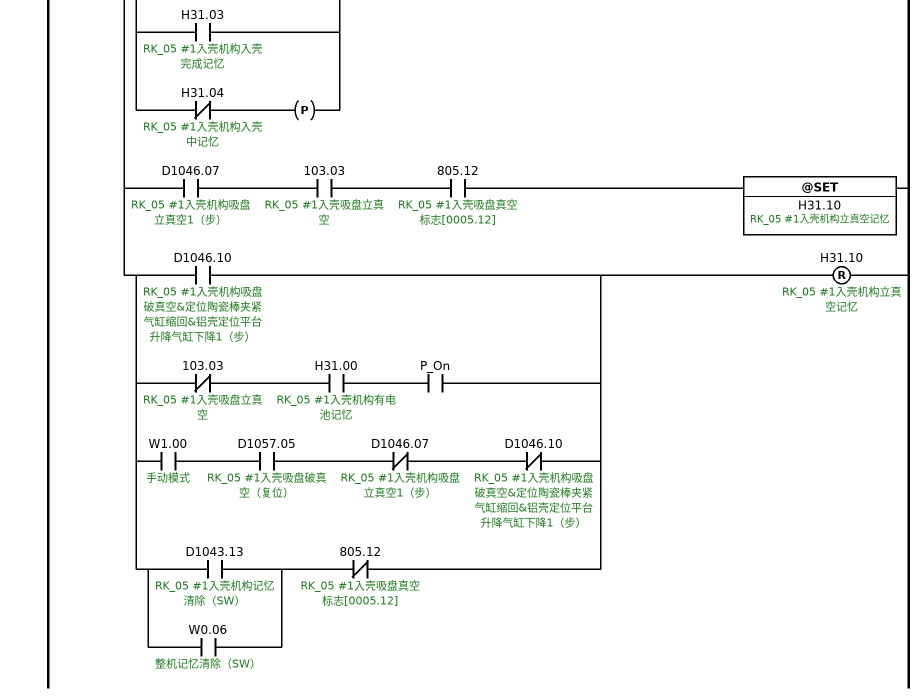
; [picture p456: 入壳_RK_05 / 自动_1入壳, rungs 30-30]
; rung 30: #1入壳机构记忆
LD P_On
OUT TR0
AND H31.03  ; RK_05 #1入壳机构入壳完成记忆
@SET H31.00  ; RK_05 #1入壳机构有电池记忆
LD TR0
LD D1092.03  ; RK_06 电池上下料机构电池下料夹爪气缸夹紧3（步）
AND H40.00  ; RK_06 U8_X 电池上下料X轴回原点记忆
AND 863.04  ; RK_06 U8_X 电池上下料X轴#1入壳取料位标志
AND 814.02  ; RK_06 电池下料升降气缸下降位标志[0014.02]
LD D1043.13  ; RK_05 #1入壳机构记忆清除（SW）
OR W0.06  ; 整机记忆清除（SW）
LDNOT 805.09  ; RK_05 #1入壳铝壳有料感应标志[0005.09]
LD H7.15  ; 空跑程序
AND 5.09  ; RK_05 #1入壳铝壳有料感应
ORLD
ANDLD
ORLD
ANDLD
RSET H31.00  ; RK_05 #1入壳机构有电池记忆
LD TR0
AND D1026.10  ; RK_03 电芯上料机构上料夹爪气缸张开（步）
LD H20.00  ; RK_03 U0_U 电芯上料X轴回原点记忆
AND 853.02  ; RK_03 U0_U 电芯上料X轴#1入壳放料位标志
AND 800.08  ; RK_03 电芯上料升降气缸下降位标志[0000.08]
LD 805.08  ; RK_05 #1入壳电芯有料感应标志[0005.08]
ANDNOT P_On
ORLD
ANDLD
@SET H31.01  ; RK_05 #1入壳机构有电芯记忆
LD TR0
LD H31.03  ; RK_05 #1入壳机构入壳完成记忆
LDNOT H31.04  ; RK_05 #1入壳机构入壳中记忆
ANDNOT 805.08  ; RK_05 #1入壳电芯有料感应标志[0005.08]
ANDNOT P_On
ORLD
LD D1043.13  ; RK_05 #1入壳机构记忆清除（SW）
OR W0.06  ; 整机记忆清除（SW）
LDNOT H31.04  ; RK_05 #1入壳机构入壳中记忆
ANDNOT 805.08  ; RK_05 #1入壳电芯有料感应标志[0005.08]
AND P_On
LD H7.15  ; 空跑程序
ANDNOT 5.08  ; RK_05 #1入壳电芯有料感应
ORLD
ANDLD
ORLD
ANDLD
RSET H31.01  ; RK_05 #1入壳机构有电芯记忆
LD TR0
AND D1089.03  ; RK_06 电池上下料机构铝壳上料夹爪气缸张开2（步）
LD H40.00  ; RK_06 U8_X 电池上下料X轴回原点记忆
AND 863.02  ; RK_06 U8_X 电池上下料X轴#1入壳放料位标志
AND 814.00  ; RK_06 铝壳上料升降气缸下降位标志[0014.00]
LD 805.09  ; RK_05 #1入壳铝壳有料感应标志[0005.09]
ANDNOT H31.00  ; RK_05 #1入壳机构有电池记忆
ORLD
ANDLD
@SET H31.02  ; RK_05 #1入壳机构有铝壳记忆
LD TR0
LD H31.03  ; RK_05 #1入壳机构入壳完成记忆
LD D1043.13  ; RK_05 #1入壳机构记忆清除（SW）
OR W0.06  ; 整机记忆清除（SW）
LDNOT 805.09  ; RK_05 #1入壳铝壳有料感应标志[0005.09]
LD H7.15  ; 空跑程序
AND 5.09  ; RK_05 #1入壳铝壳有料感应
ORLD
ANDLD
ORLD
ANDLD
RSET H31.02  ; RK_05 #1入壳机构有铝壳记忆
LD TR0
AND D1049.08  ; RK_05 #1入壳机构Y轴入壳位2（步）
AND 854.03  ; RK_05 U2_X #1入壳Y轴入壳位标志
AND H30.00  ; RK_05 U2_X #1入壳Y轴回原点记忆
ANDNOT W421.00  ; RK_05 #1入壳压力高[alm]
@SET H31.03  ; RK_05 #1入壳机构入壳完成记忆
LD TR0
LD H31.00  ; RK_05 #1入壳机构有电池记忆
LD D1043.13  ; RK_05 #1入壳机构记忆清除（SW）
OR W0.06  ; 整机记忆清除（SW）
LDNOT 805.09  ; RK_05 #1入壳铝壳有料感应标志[0005.09]
LD H7.15  ; 空跑程序
AND 5.09  ; RK_05 #1入壳铝壳有料感应
ORLD
ANDLD
ORLD
ANDLD
RSET H31.03  ; RK_05 #1入壳机构入壳完成记忆
LD TR0
AND D1049.02  ; RK_05 #1入壳机构Y轴电芯定位夹爪气缸松开位2（步）
@SET H31.04  ; RK_05 #1入壳机构入壳中记忆
LD TR0
LD H31.03  ; RK_05 #1入壳机构入壳完成记忆
LD D1043.13  ; RK_05 #1入壳机构记忆清除（SW）
OR W0.06  ; 整机记忆清除（SW）
LDNOT 805.09  ; RK_05 #1入壳铝壳有料感应标志[0005.09]
LD H7.15  ; 空跑程序
AND 5.09  ; RK_05 #1入壳铝壳有料感应
ORLD
ANDLD
ORLD
ANDLD
RSET H31.04  ; RK_05 #1入壳机构入壳中记忆
LD TR0
AND D1049.04  ; RK_05 #1入壳机构Y轴滚轮压紧位2（步）
AND 854.01  ; RK_05 U2_X #1入壳Y轴滚轮压紧位标志
@SET H31.06  ; RK_05 #1入壳机构Y轴滚轮压紧位记忆
LD TR0
LD D1049.06  ; RK_05 #1入壳机构Y轴滚轮松开位2（步）
OR H31.03  ; RK_05 #1入壳机构入壳完成记忆
ORNOT H31.04  ; RK_05 #1入壳机构入壳中记忆
ANDLD
RSET H31.06  ; RK_05 #1入壳机构Y轴滚轮压紧位记忆
LD TR0
AND D1049.06  ; RK_05 #1入壳机构Y轴滚轮松开位2（步）
AND 854.02  ; RK_05 U2_X #1入壳Y轴滚轮松开位标志
@SET H31.07  ; RK_05 #1入壳机构Y轴滚轮松开位记忆
LD TR0
LD H31.03  ; RK_05 #1入壳机构入壳完成记忆
ORNOT H31.04  ; RK_05 #1入壳机构入壳中记忆
ANDLD
RSET H31.07  ; RK_05 #1入壳机构Y轴滚轮松开位记忆
LD TR0
AND D1049.02  ; RK_05 #1入壳机构Y轴电芯定位夹爪气缸松开位2（步）
AND 854.04  ; RK_05 U2_X #1入壳Y轴电芯定位夹爪松开位标志
@SET H31.09  ; RK_05 #1入壳机构Y轴电芯定位夹爪松开位记忆
LD TR0
LD D1049.04  ; RK_05 #1入壳机构Y轴滚轮压紧位2（步）
OR H31.06  ; RK_05 #1入壳机构Y轴滚轮压紧位记忆
OR H31.03  ; RK_05 #1入壳机构入壳完成记忆
LDNOT H31.04  ; RK_05 #1入壳机构入壳中记忆
UP(521)
ORLD
ANDLD
RSET H31.09  ; RK_05 #1入壳机构Y轴电芯定位夹爪松开位记忆
LD TR0
AND D1046.07  ; RK_05 #1入壳机构吸盘立真空1（步）
AND 103.03  ; RK_05 #1入壳吸盘立真空
AND 805.12  ; RK_05 #1入壳吸盘真空标志[0005.12]
@SET H31.10  ; RK_05 #1入壳机构立真空记忆
LD TR0
LD D1046.10  ; RK_05 #1入壳机构吸盘破真空&定位陶瓷棒夹紧气缸缩回&铝壳定位平台升降气缸下降1（步）
LDNOT 103.03  ; RK_05 #1入壳吸盘立真空
AND H31.00  ; RK_05 #1入壳机构有电池记忆
AND P_On
ORLD
LD W1.00  ; 手动模式  // 20181116新增
AND D1057.05  ; RK_05 #1入壳吸盘破真空（复位）
ANDNOT D1046.07  ; RK_05 #1入壳机构吸盘立真空1（步）
ANDNOT D1046.10  ; RK_05 #1入壳机构吸盘破真空&定位陶瓷棒夹紧气缸缩回&铝壳定位平台升降气缸下降1（步）
ORLD
LD D1043.13  ; RK_05 #1入壳机构记忆清除（SW）
OR W0.06  ; 整机记忆清除（SW）
ANDNOT 805.12  ; RK_05 #1入壳吸盘真空标志[0005.12]
ORLD
ANDLD
RSET H31.10  ; RK_05 #1入壳机构立真空记忆

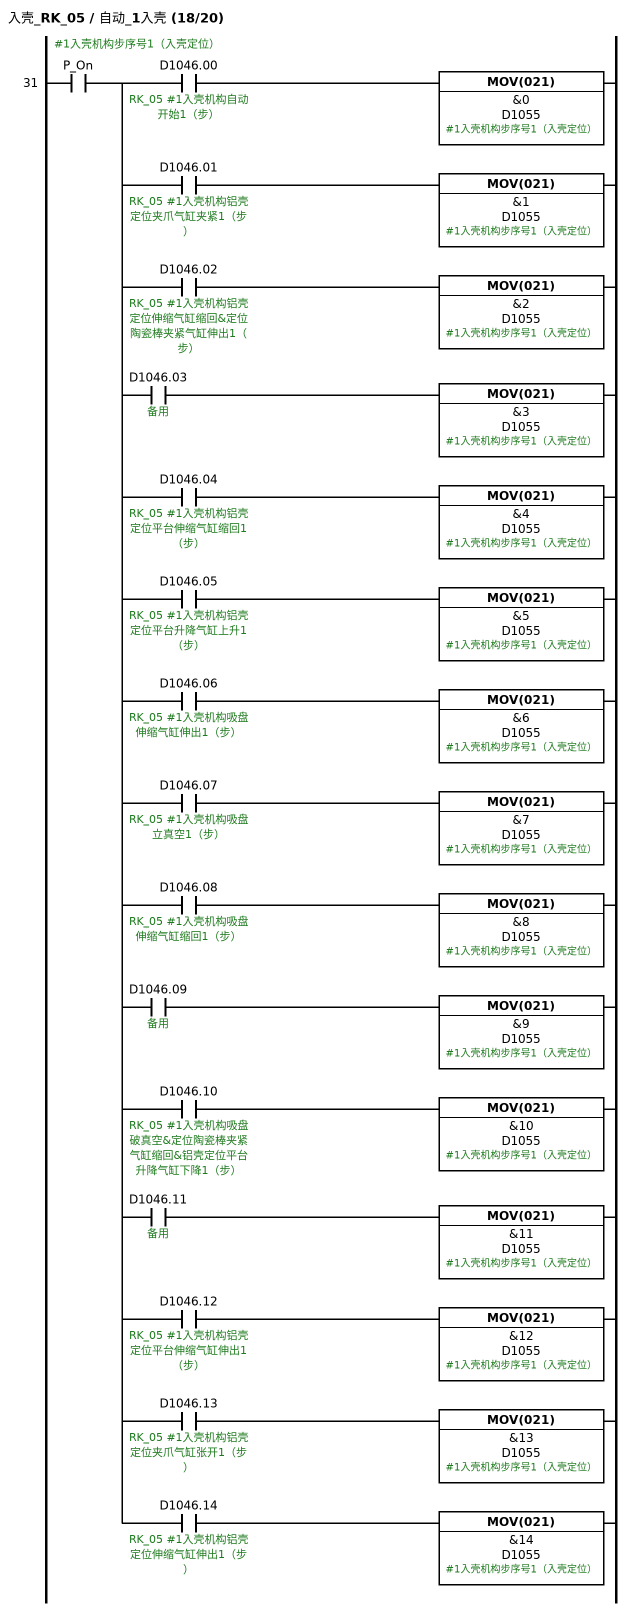
; rung 31: #1入壳机构步序号1（入壳定位）
LD P_On
OUT TR0
AND D1046.00  ; RK_05 #1入壳机构自动开始1（步）
MOV(021) &0 D1055  ; #1入壳机构步序号1（入壳定位）
LD TR0
AND D1046.01  ; RK_05 #1入壳机构铝壳定位夹爪气缸夹紧1（步）
MOV(021) &1 D1055  ; #1入壳机构步序号1（入壳定位）
LD TR0
AND D1046.02  ; RK_05 #1入壳机构铝壳定位伸缩气缸缩回&定位陶瓷棒夹紧气缸伸出1（步）
MOV(021) &2 D1055  ; #1入壳机构步序号1（入壳定位）
LD TR0
AND D1046.03  ; 备用
MOV(021) &3 D1055  ; #1入壳机构步序号1（入壳定位）
LD TR0
AND D1046.04  ; RK_05 #1入壳机构铝壳定位平台伸缩气缸缩回1（步）
MOV(021) &4 D1055  ; #1入壳机构步序号1（入壳定位）
LD TR0
AND D1046.05  ; RK_05 #1入壳机构铝壳定位平台升降气缸上升1（步）
MOV(021) &5 D1055  ; #1入壳机构步序号1（入壳定位）
LD TR0
AND D1046.06  ; RK_05 #1入壳机构吸盘伸缩气缸伸出1（步）
MOV(021) &6 D1055  ; #1入壳机构步序号1（入壳定位）
LD TR0
AND D1046.07  ; RK_05 #1入壳机构吸盘立真空1（步）
MOV(021) &7 D1055  ; #1入壳机构步序号1（入壳定位）
LD TR0
AND D1046.08  ; RK_05 #1入壳机构吸盘伸缩气缸缩回1（步）
MOV(021) &8 D1055  ; #1入壳机构步序号1（入壳定位）
LD TR0
AND D1046.09  ; 备用
MOV(021) &9 D1055  ; #1入壳机构步序号1（入壳定位）
LD TR0
AND D1046.10  ; RK_05 #1入壳机构吸盘破真空&定位陶瓷棒夹紧气缸缩回&铝壳定位平台升降气缸下降1（步）
MOV(021) &10 D1055  ; #1入壳机构步序号1（入壳定位）
LD TR0
AND D1046.11  ; 备用
MOV(021) &11 D1055  ; #1入壳机构步序号1（入壳定位）
LD TR0
AND D1046.12  ; RK_05 #1入壳机构铝壳定位平台伸缩气缸伸出1（步）
MOV(021) &12 D1055  ; #1入壳机构步序号1（入壳定位）
LD TR0
AND D1046.13  ; RK_05 #1入壳机构铝壳定位夹爪气缸张开1（步）
MOV(021) &13 D1055  ; #1入壳机构步序号1（入壳定位）
LD TR0
AND D1046.14  ; RK_05 #1入壳机构铝壳定位伸缩气缸伸出1（步）
MOV(021) &14 D1055  ; #1入壳机构步序号1（入壳定位）

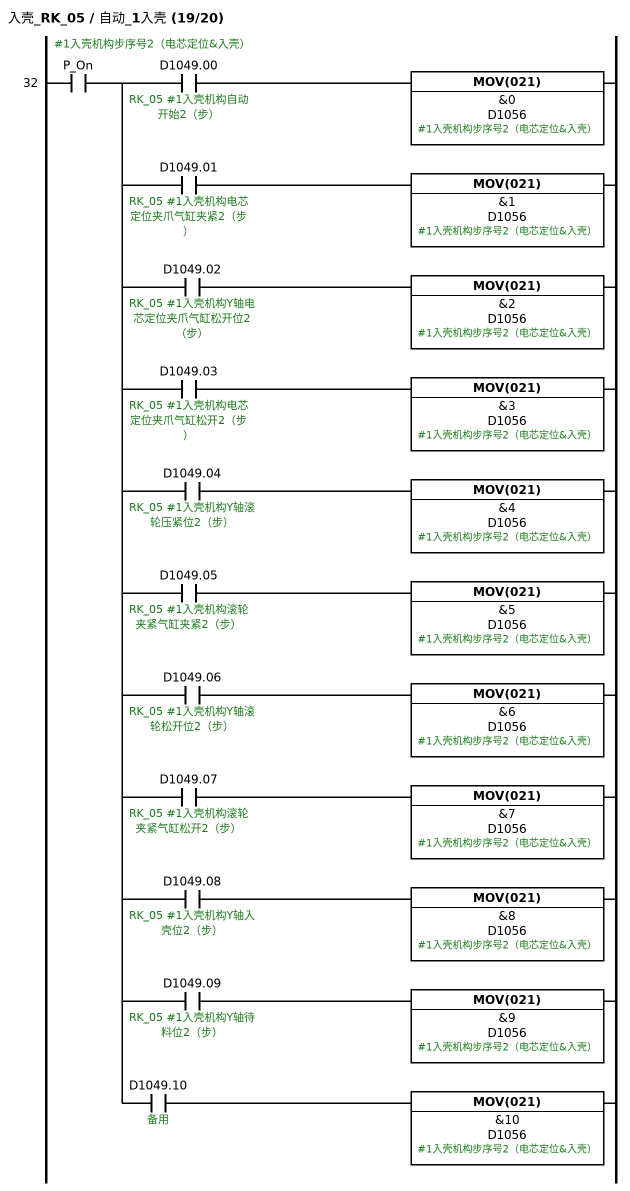
; rung 32: #1入壳机构步序号2（电芯定位&入壳）
LD P_On
OUT TR0
AND D1049.00  ; RK_05 #1入壳机构自动开始2（步）
MOV(021) &0 D1056  ; #1入壳机构步序号2（电芯定位&入壳）
LD TR0
AND D1049.01  ; RK_05 #1入壳机构电芯定位夹爪气缸夹紧2（步）
MOV(021) &1 D1056  ; #1入壳机构步序号2（电芯定位&入壳）
LD TR0
AND D1049.02  ; RK_05 #1入壳机构Y轴电芯定位夹爪气缸松开位2（步）
MOV(021) &2 D1056  ; #1入壳机构步序号2（电芯定位&入壳）
LD TR0
AND D1049.03  ; RK_05 #1入壳机构电芯定位夹爪气缸松开2（步）
MOV(021) &3 D1056  ; #1入壳机构步序号2（电芯定位&入壳）
LD TR0
AND D1049.04  ; RK_05 #1入壳机构Y轴滚轮压紧位2（步）
MOV(021) &4 D1056  ; #1入壳机构步序号2（电芯定位&入壳）
LD TR0
AND D1049.05  ; RK_05 #1入壳机构滚轮夹紧气缸夹紧2（步）
MOV(021) &5 D1056  ; #1入壳机构步序号2（电芯定位&入壳）
LD TR0
AND D1049.06  ; RK_05 #1入壳机构Y轴滚轮松开位2（步）
MOV(021) &6 D1056  ; #1入壳机构步序号2（电芯定位&入壳）
LD TR0
AND D1049.07  ; RK_05 #1入壳机构滚轮夹紧气缸松开2（步）
MOV(021) &7 D1056  ; #1入壳机构步序号2（电芯定位&入壳）
LD TR0
AND D1049.08  ; RK_05 #1入壳机构Y轴入壳位2（步）
MOV(021) &8 D1056  ; #1入壳机构步序号2（电芯定位&入壳）
LD TR0
AND D1049.09  ; RK_05 #1入壳机构Y轴待料位2（步）
MOV(021) &9 D1056  ; #1入壳机构步序号2（电芯定位&入壳）
LD TR0
AND D1049.10  ; 备用
MOV(021) &10 D1056  ; #1入壳机构步序号2（电芯定位&入壳）

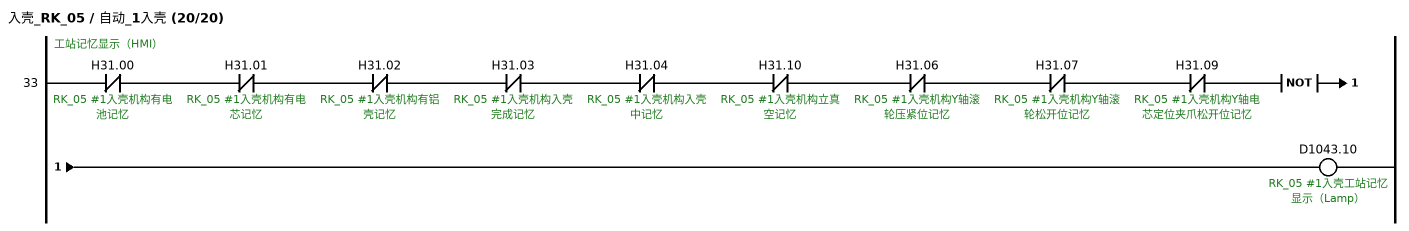
; rung 33: 工站记忆显示（HMI）
LDNOT H31.00  ; RK_05 #1入壳机构有电池记忆
ANDNOT H31.01  ; RK_05 #1入壳机构有电芯记忆
ANDNOT H31.02  ; RK_05 #1入壳机构有铝壳记忆
ANDNOT H31.03  ; RK_05 #1入壳机构入壳完成记忆
ANDNOT H31.04  ; RK_05 #1入壳机构入壳中记忆
ANDNOT H31.10  ; RK_05 #1入壳机构立真空记忆
ANDNOT H31.06  ; RK_05 #1入壳机构Y轴滚轮压紧位记忆
ANDNOT H31.07  ; RK_05 #1入壳机构Y轴滚轮松开位记忆
ANDNOT H31.09  ; RK_05 #1入壳机构Y轴电芯定位夹爪松开位记忆
NOT(520)
OUT D1043.10  ; RK_05 #1入壳工站记忆显示（Lamp）

### Section 自动_2入壳

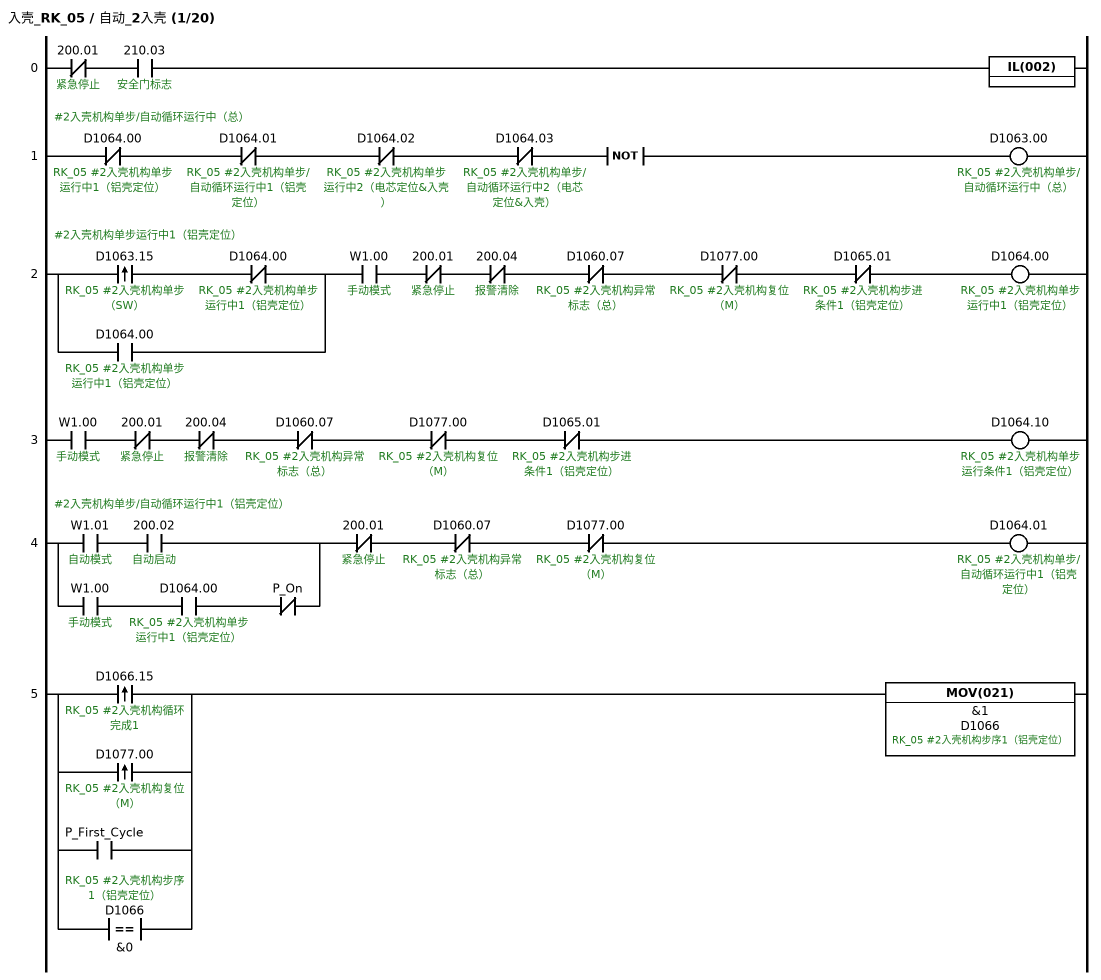
; rung 0
LDNOT 200.01  ; 紧急停止
AND 210.03  ; 安全门标志
IL(002)
; rung 1: #2入壳机构单步/自动循环运行中（总）
LDNOT D1064.00  ; RK_05 #2入壳机构单步运行中1（铝壳定位）
ANDNOT D1064.01  ; RK_05 #2入壳机构单步/自动循环运行中1（铝壳定位）
ANDNOT D1064.02  ; RK_05 #2入壳机构单步运行中2（电芯定位&入壳）
ANDNOT D1064.03  ; RK_05 #2入壳机构单步/自动循环运行中2（电芯定位&入壳）
NOT(520)
OUT D1063.00  ; RK_05 #2入壳机构单步/自动循环运行中（总）
; rung 2: #2入壳机构单步运行中1（铝壳定位）
@LD D1063.15  ; RK_05 #2入壳机构单步（SW）
ANDNOT D1064.00  ; RK_05 #2入壳机构单步运行中1（铝壳定位）
OR D1064.00  ; RK_05 #2入壳机构单步运行中1（铝壳定位）
AND W1.00  ; 手动模式
ANDNOT 200.01  ; 紧急停止
ANDNOT 200.04  ; 报警清除
ANDNOT D1060.07  ; RK_05 #2入壳机构异常标志（总）
ANDNOT D1077.00  ; RK_05 #2入壳机构复位（M）
ANDNOT D1065.01  ; RK_05 #2入壳机构步进条件1（铝壳定位）
OUT D1064.00  ; RK_05 #2入壳机构单步运行中1（铝壳定位）
; rung 3
LD W1.00  ; 手动模式
ANDNOT 200.01  ; 紧急停止
ANDNOT 200.04  ; 报警清除
ANDNOT D1060.07  ; RK_05 #2入壳机构异常标志（总）
ANDNOT D1077.00  ; RK_05 #2入壳机构复位（M）
ANDNOT D1065.01  ; RK_05 #2入壳机构步进条件1（铝壳定位）
OUT D1064.10  ; RK_05 #2入壳机构单步运行条件1（铝壳定位）
; rung 4: #2入壳机构单步/自动循环运行中1（铝壳定位）
LD W1.01  ; 自动模式
AND 200.02  ; 自动启动
LD W1.00  ; 手动模式
AND D1064.00  ; RK_05 #2入壳机构单步运行中1（铝壳定位）
ANDNOT P_On
ORLD
ANDNOT 200.01  ; 紧急停止
ANDNOT D1060.07  ; RK_05 #2入壳机构异常标志（总）
ANDNOT D1077.00  ; RK_05 #2入壳机构复位（M）
OUT D1064.01  ; RK_05 #2入壳机构单步/自动循环运行中1（铝壳定位）
; rung 5
@LD D1066.15  ; RK_05 #2入壳机构循环完成1
@OR D1077.00  ; RK_05 #2入壳机构复位（M）
OR P_First_Cycle
OR=(300) D1066 &0  ; RK_05 #2入壳机构步序1（铝壳定位）
MOV(021) &1 D1066  ; RK_05 #2入壳机构步序1（铝壳定位）

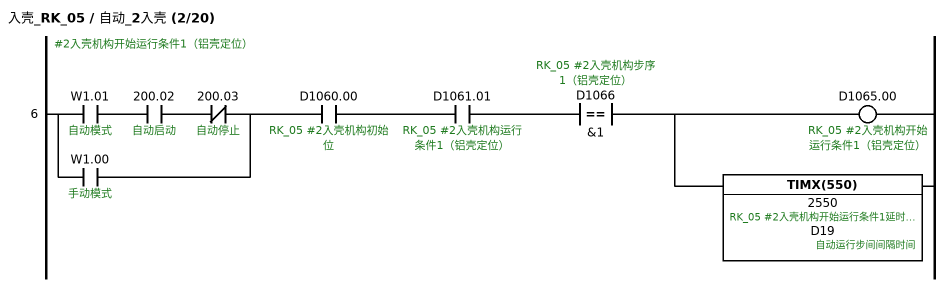
; rung 6: #2入壳机构开始运行条件1（铝壳定位）
LD W1.01  ; 自动模式
AND 200.02  ; 自动启动
ANDNOT 200.03  ; 自动停止
OR W1.00  ; 手动模式
AND D1060.00  ; RK_05 #2入壳机构初始位
AND D1061.01  ; RK_05 #2入壳机构运行条件1（铝壳定位）
AND=(300) D1066 &1  ; RK_05 #2入壳机构步序1（铝壳定位）
OUT D1065.00  ; RK_05 #2入壳机构开始运行条件1（铝壳定位）
TIMX(550) 2550 D19  ; 自动运行步间间隔时间, RK_05 #2入壳机构开始运行条件1延时（铝壳定位）

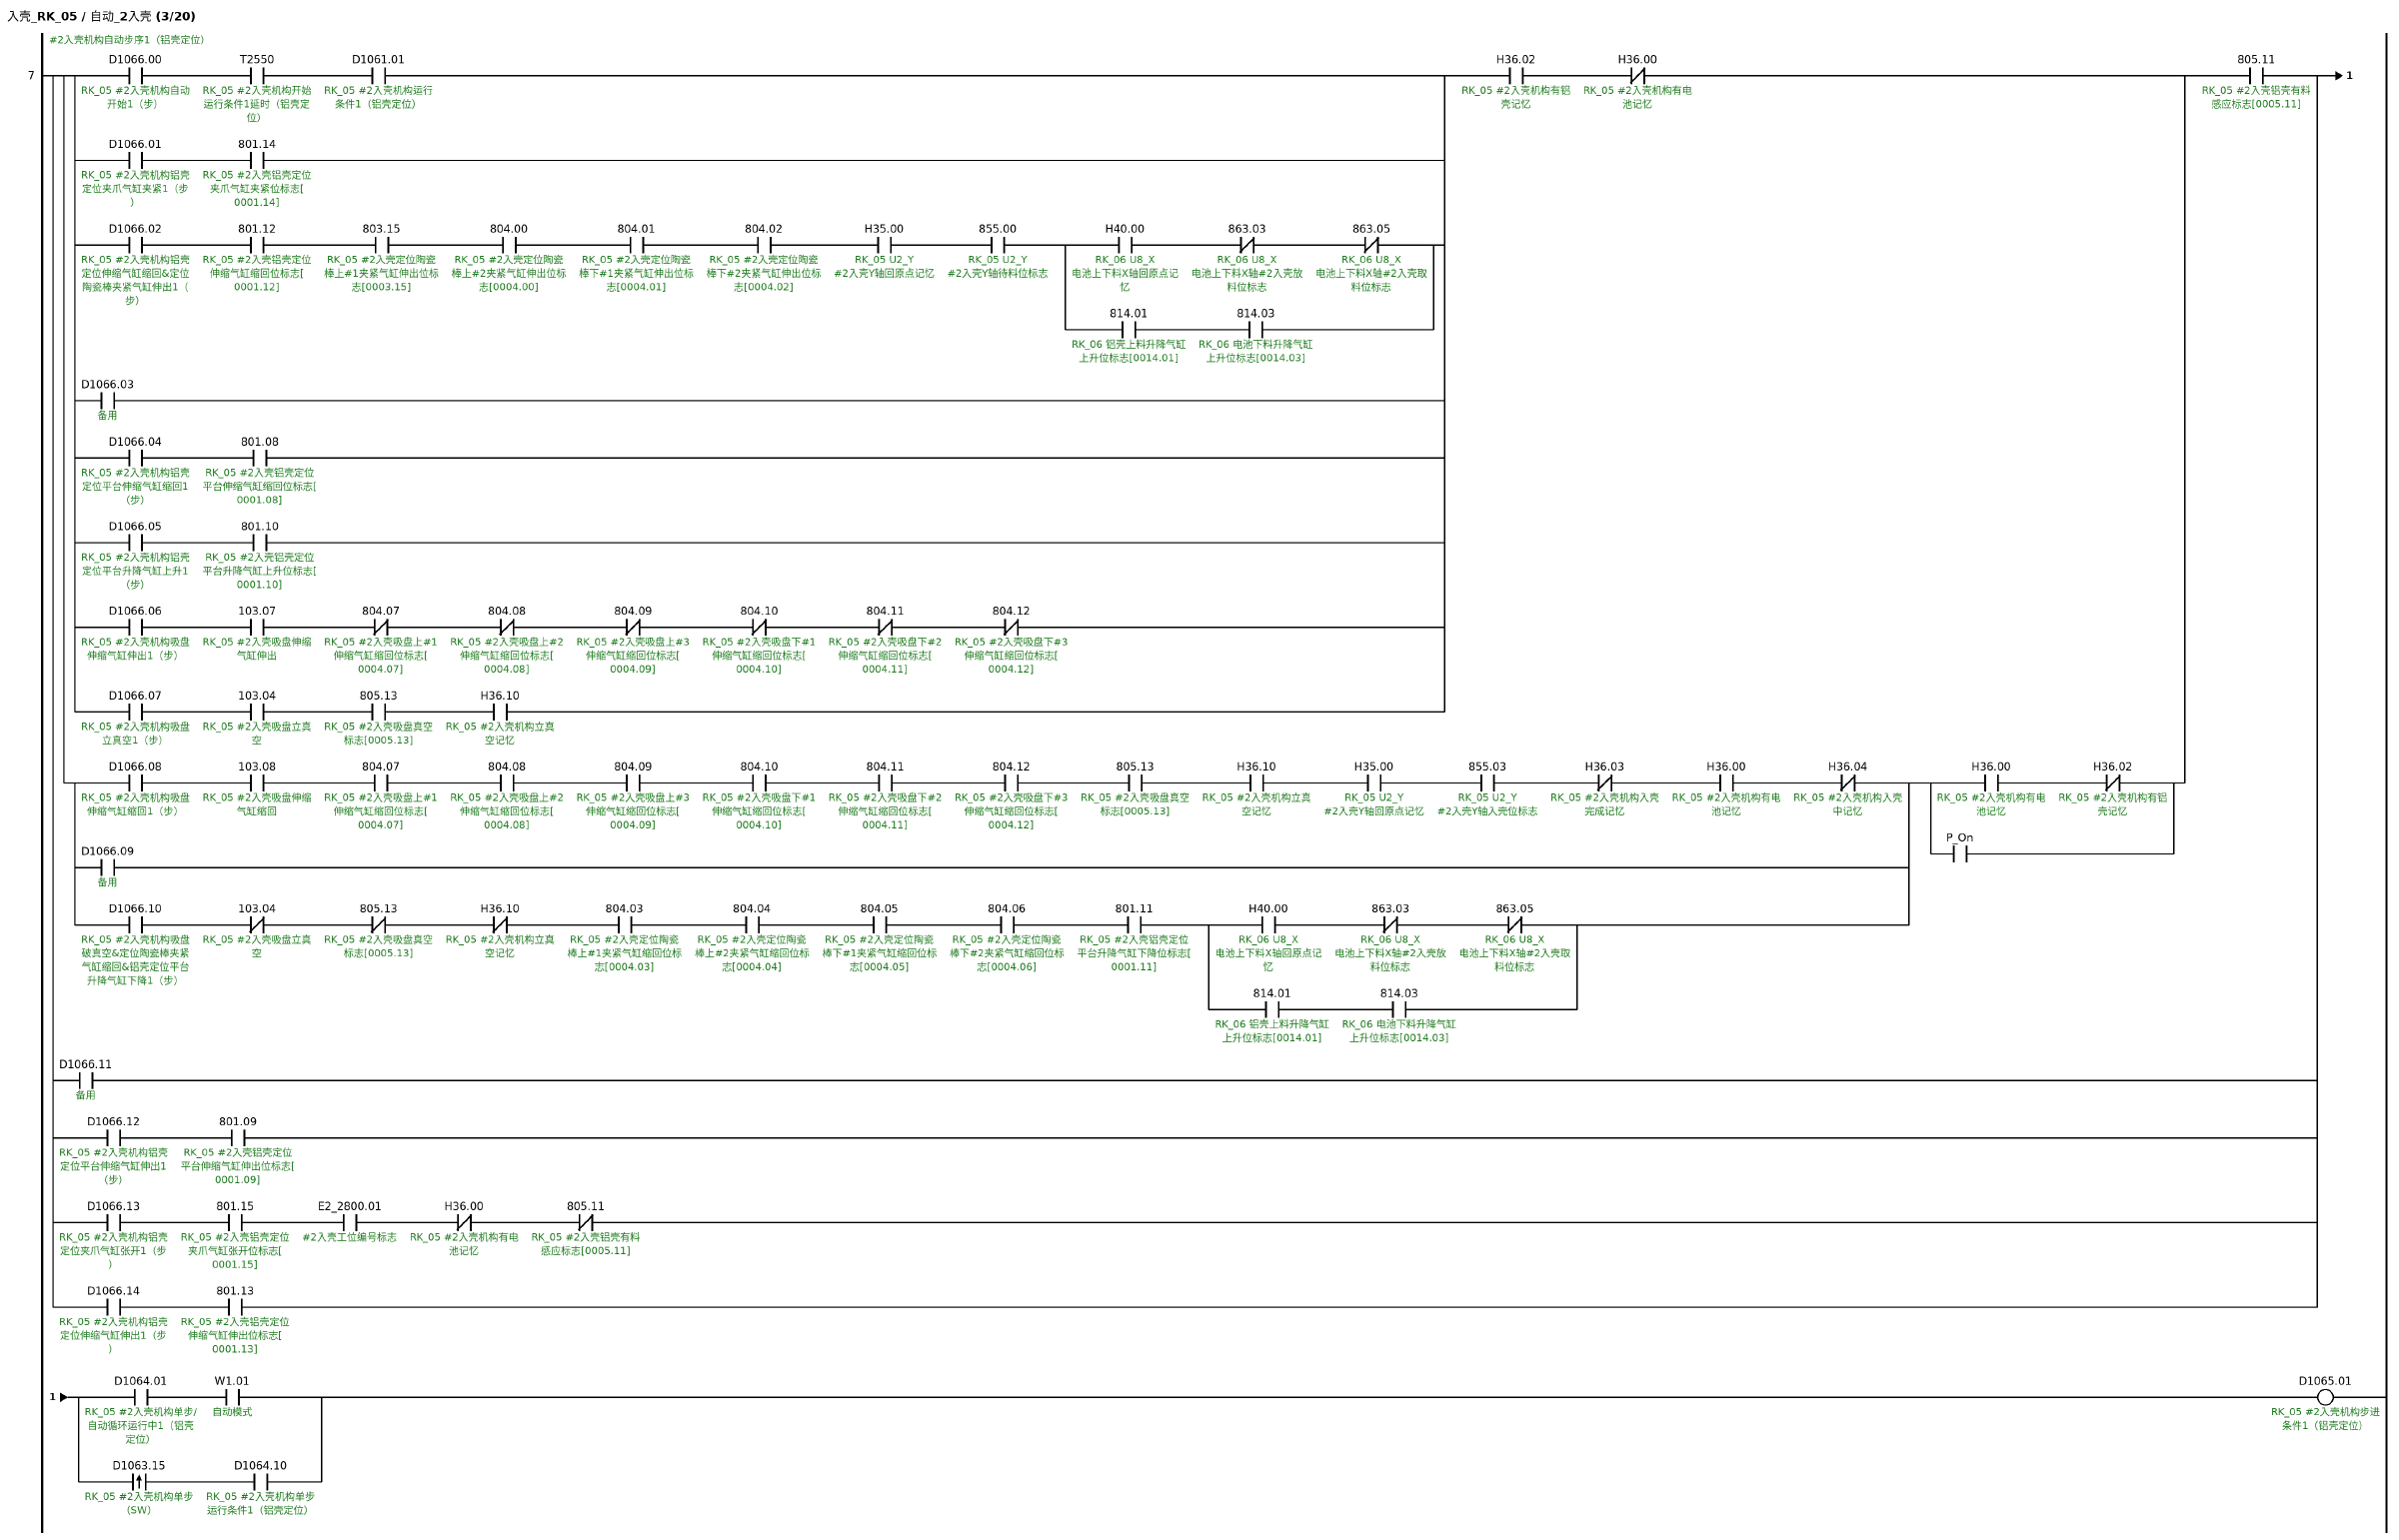
; rung 7: #2入壳机构自动步序1（铝壳定位）
LD D1066.00  ; RK_05 #2入壳机构自动开始1（步）
AND T2550  ; RK_05 #2入壳机构开始运行条件1延时（铝壳定位）
AND D1061.01  ; RK_05 #2入壳机构运行条件1（铝壳定位）
LD D1066.01  ; RK_05 #2入壳机构铝壳定位夹爪气缸夹紧1（步）
AND 801.14  ; RK_05 #2入壳铝壳定位夹爪气缸夹紧位标志[0001.14]
ORLD
LD D1066.02  ; RK_05 #2入壳机构铝壳定位伸缩气缸缩回&定位陶瓷棒夹紧气缸伸出1（步）
AND 801.12  ; RK_05 #2入壳铝壳定位伸缩气缸缩回位标志[0001.12]
AND 803.15  ; RK_05 #2入壳定位陶瓷棒上#1夹紧气缸伸出位标志[0003.15]
AND 804.00  ; RK_05 #2入壳定位陶瓷棒上#2夹紧气缸伸出位标志[0004.00]
AND 804.01  ; RK_05 #2入壳定位陶瓷棒下#1夹紧气缸伸出位标志[0004.01]
AND 804.02  ; RK_05 #2入壳定位陶瓷棒下#2夹紧气缸伸出位标志[0004.02]
AND H35.00  ; RK_05 U2_Y #2入壳Y轴回原点记忆
AND 855.00  ; RK_05 U2_Y #2入壳Y轴待料位标志
LD H40.00  ; RK_06 U8_X 电池上下料X轴回原点记忆
ANDNOT 863.03  ; RK_06 U8_X 电池上下料X轴#2入壳放料位标志
ANDNOT 863.05  ; RK_06 U8_X 电池上下料X轴#2入壳取料位标志
LD 814.01  ; RK_06 铝壳上料升降气缸上升位标志[0014.01]
AND 814.03  ; RK_06 电池下料升降气缸上升位标志[0014.03]
ORLD
ANDLD
ORLD
OR D1066.03  ; 备用
LD D1066.04  ; RK_05 #2入壳机构铝壳定位平台伸缩气缸缩回1（步）
AND 801.08  ; RK_05 #2入壳铝壳定位平台伸缩气缸缩回位标志[0001.08]
ORLD
LD D1066.05  ; RK_05 #2入壳机构铝壳定位平台升降气缸上升1（步）
AND 801.10  ; RK_05 #2入壳铝壳定位平台升降气缸上升位标志[0001.10]
ORLD
LD D1066.06  ; RK_05 #2入壳机构吸盘伸缩气缸伸出1（步）
AND 103.07  ; RK_05 #2入壳吸盘伸缩气缸伸出
ANDNOT 804.07  ; RK_05 #2入壳吸盘上#1伸缩气缸缩回位标志[0004.07]
ANDNOT 804.08  ; RK_05 #2入壳吸盘上#2伸缩气缸缩回位标志[0004.08]
ANDNOT 804.09  ; RK_05 #2入壳吸盘上#3伸缩气缸缩回位标志[0004.09]
ANDNOT 804.10  ; RK_05 #2入壳吸盘下#1伸缩气缸缩回位标志[0004.10]
ANDNOT 804.11  ; RK_05 #2入壳吸盘下#2伸缩气缸缩回位标志[0004.11]
ANDNOT 804.12  ; RK_05 #2入壳吸盘下#3伸缩气缸缩回位标志[0004.12]
ORLD
LD D1066.07  ; RK_05 #2入壳机构吸盘立真空1（步）
AND 103.04  ; RK_05 #2入壳吸盘立真空
AND 805.13  ; RK_05 #2入壳吸盘真空标志[0005.13]
AND H36.10  ; RK_05 #2入壳机构立真空记忆
ORLD
AND H36.02  ; RK_05 #2入壳机构有铝壳记忆
ANDNOT H36.00  ; RK_05 #2入壳机构有电池记忆
LD D1066.08  ; RK_05 #2入壳机构吸盘伸缩气缸缩回1（步）
AND 103.08  ; RK_05 #2入壳吸盘伸缩气缸缩回
AND 804.07  ; RK_05 #2入壳吸盘上#1伸缩气缸缩回位标志[0004.07]
AND 804.08  ; RK_05 #2入壳吸盘上#2伸缩气缸缩回位标志[0004.08]
AND 804.09  ; RK_05 #2入壳吸盘上#3伸缩气缸缩回位标志[0004.09]
AND 804.10  ; RK_05 #2入壳吸盘下#1伸缩气缸缩回位标志[0004.10]
AND 804.11  ; RK_05 #2入壳吸盘下#2伸缩气缸缩回位标志[0004.11]
AND 804.12  ; RK_05 #2入壳吸盘下#3伸缩气缸缩回位标志[0004.12]
AND 805.13  ; RK_05 #2入壳吸盘真空标志[0005.13]
AND H36.10  ; RK_05 #2入壳机构立真空记忆
AND H35.00  ; RK_05 U2_Y #2入壳Y轴回原点记忆
AND 855.03  ; RK_05 U2_Y #2入壳Y轴入壳位标志
ANDNOT H36.03  ; RK_05 #2入壳机构入壳完成记忆
AND H36.00  ; RK_05 #2入壳机构有电池记忆
ANDNOT H36.04  ; RK_05 #2入壳机构入壳中记忆
OR D1066.09  ; 备用
LD D1066.10  ; RK_05 #2入壳机构吸盘破真空&定位陶瓷棒夹紧气缸缩回&铝壳定位平台升降气缸下降1（步）
ANDNOT 103.04  ; RK_05 #2入壳吸盘立真空
ANDNOT 805.13  ; RK_05 #2入壳吸盘真空标志[0005.13]
ANDNOT H36.10  ; RK_05 #2入壳机构立真空记忆
AND 804.03  ; RK_05 #2入壳定位陶瓷棒上#1夹紧气缸缩回位标志[0004.03]
AND 804.04  ; RK_05 #2入壳定位陶瓷棒上#2夹紧气缸缩回位标志[0004.04]
AND 804.05  ; RK_05 #2入壳定位陶瓷棒下#1夹紧气缸缩回位标志[0004.05]
AND 804.06  ; RK_05 #2入壳定位陶瓷棒下#2夹紧气缸缩回位标志[0004.06]
AND 801.11  ; RK_05 #2入壳铝壳定位平台升降气缸下降位标志[0001.11]
LD H40.00  ; RK_06 U8_X 电池上下料X轴回原点记忆
ANDNOT 863.03  ; RK_06 U8_X 电池上下料X轴#2入壳放料位标志
ANDNOT 863.05  ; RK_06 U8_X 电池上下料X轴#2入壳取料位标志
LD 814.01  ; RK_06 铝壳上料升降气缸上升位标志[0014.01]
AND 814.03  ; RK_06 电池下料升降气缸上升位标志[0014.03]
ORLD
ANDLD
ORLD
LD H36.00  ; RK_05 #2入壳机构有电池记忆
ANDNOT H36.02  ; RK_05 #2入壳机构有铝壳记忆
OR P_On
ANDLD
ORLD
AND 805.11  ; RK_05 #2入壳铝壳有料感应标志[0005.11]
OR D1066.11  ; 备用
LD D1066.12  ; RK_05 #2入壳机构铝壳定位平台伸缩气缸伸出1（步）
AND 801.09  ; RK_05 #2入壳铝壳定位平台伸缩气缸伸出位标志[0001.09]
ORLD
LD D1066.13  ; RK_05 #2入壳机构铝壳定位夹爪气缸张开1（步）
AND 801.15  ; RK_05 #2入壳铝壳定位夹爪气缸张开位标志[0001.15]
AND E2_2800.01  ; #2入壳工位编号标志
ANDNOT H36.00  ; RK_05 #2入壳机构有电池记忆
ANDNOT 805.11  ; RK_05 #2入壳铝壳有料感应标志[0005.11]
ORLD
LD D1066.14  ; RK_05 #2入壳机构铝壳定位伸缩气缸伸出1（步）
AND 801.13  ; RK_05 #2入壳铝壳定位伸缩气缸伸出位标志[0001.13]
ORLD
LD D1064.01  ; RK_05 #2入壳机构单步/自动循环运行中1（铝壳定位）
AND W1.01  ; 自动模式
@LD D1063.15  ; RK_05 #2入壳机构单步（SW）
AND D1064.10  ; RK_05 #2入壳机构单步运行条件1（铝壳定位）
ORLD
ANDLD
OUT D1065.01  ; RK_05 #2入壳机构步进条件1（铝壳定位）

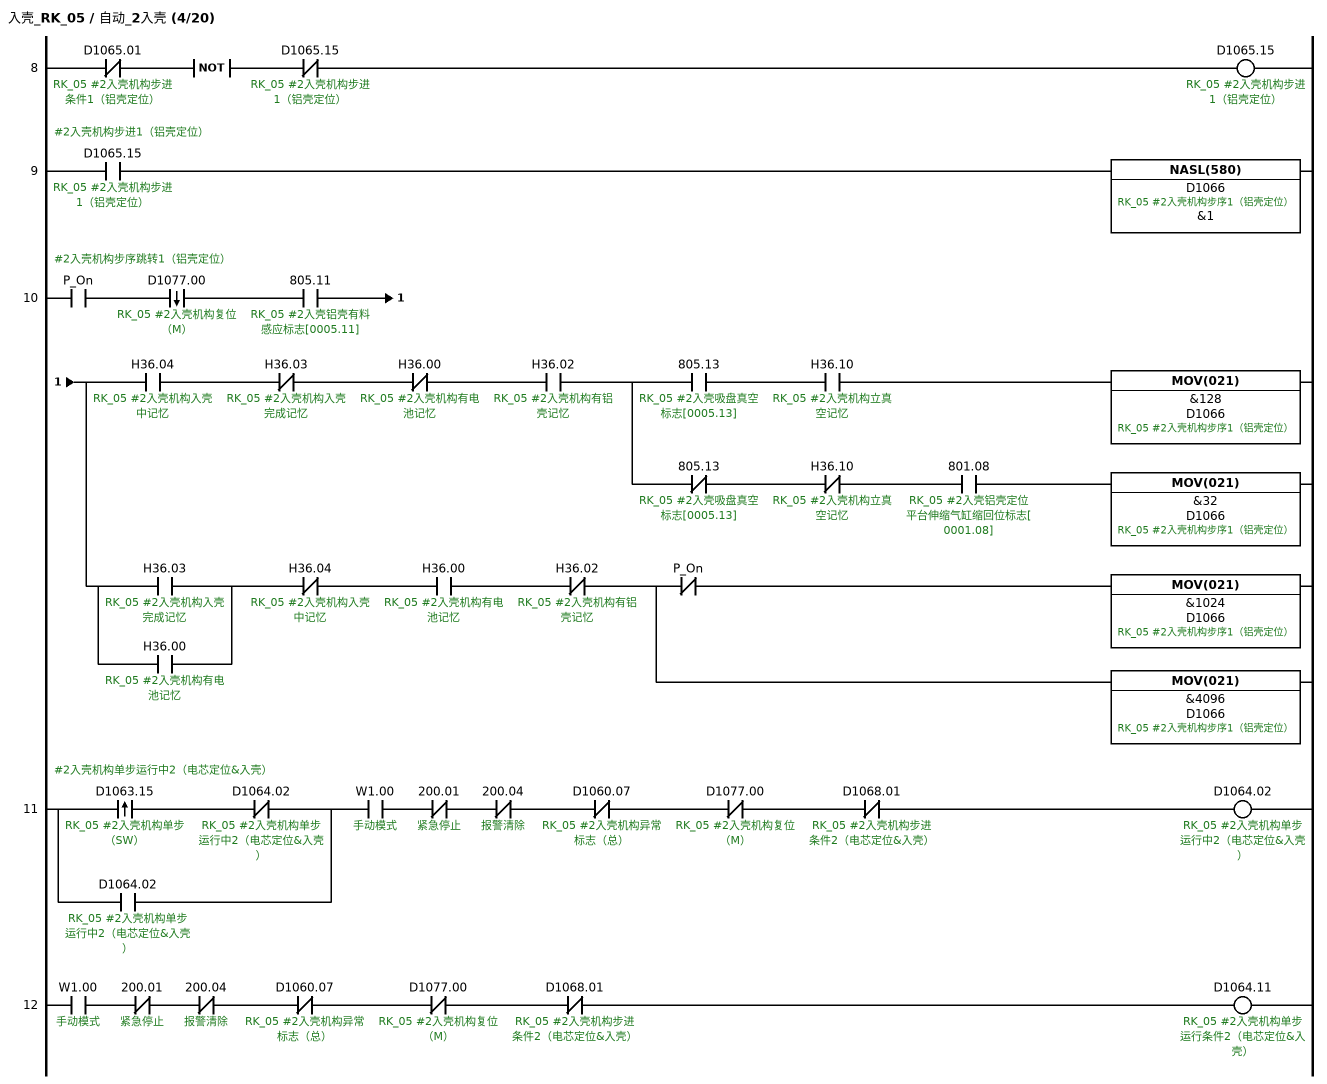
; rung 8
LDNOT D1065.01  ; RK_05 #2入壳机构步进条件1（铝壳定位）
NOT(520)
ANDNOT D1065.15  ; RK_05 #2入壳机构步进1（铝壳定位）
OUT D1065.15  ; RK_05 #2入壳机构步进1（铝壳定位）
; rung 9: #2入壳机构步进1（铝壳定位）
LD D1065.15  ; RK_05 #2入壳机构步进1（铝壳定位）
NASL(580) D1066 &1  ; RK_05 #2入壳机构步序1（铝壳定位）
; rung 10: #2入壳机构步序跳转1（铝壳定位）
LD P_On
%AND D1077.00  ; RK_05 #2入壳机构复位（M）
AND 805.11  ; RK_05 #2入壳铝壳有料感应标志[0005.11]
OUT TR0
AND H36.04  ; RK_05 #2入壳机构入壳中记忆
ANDNOT H36.03  ; RK_05 #2入壳机构入壳完成记忆
ANDNOT H36.00  ; RK_05 #2入壳机构有电池记忆
AND H36.02  ; RK_05 #2入壳机构有铝壳记忆
OUT TR1
AND 805.13  ; RK_05 #2入壳吸盘真空标志[0005.13]
AND H36.10  ; RK_05 #2入壳机构立真空记忆
MOV(021) &128 D1066  ; RK_05 #2入壳机构步序1（铝壳定位）  // RK_05 #2入壳机构吸盘立真空1步（D1066.07）
LD TR1
ANDNOT 805.13  ; RK_05 #2入壳吸盘真空标志[0005.13]
ANDNOT H36.10  ; RK_05 #2入壳机构立真空记忆
AND 801.08  ; RK_05 #2入壳铝壳定位平台伸缩气缸缩回位标志[0001.08]
MOV(021) &32 D1066  ; RK_05 #2入壳机构步序1（铝壳定位）  // RK_05 #2入壳机构铝壳定位平台升降气缸上升1步（D1066.05）
LD TR0
LD H36.03  ; RK_05 #2入壳机构入壳完成记忆
OR H36.00  ; RK_05 #2入壳机构有电池记忆
ANDLD
ANDNOT H36.04  ; RK_05 #2入壳机构入壳中记忆
AND H36.00  ; RK_05 #2入壳机构有电池记忆
ANDNOT H36.02  ; RK_05 #2入壳机构有铝壳记忆
OUT TR0
ANDNOT P_On
MOV(021) &1024 D1066  ; RK_05 #2入壳机构步序1（铝壳定位）  // RK_05 #2入壳机构吸盘破真空&定位陶瓷棒夹紧气缸缩回&铝壳定位平台升降气缸下降1步（D1066.10）
LD TR0
MOV(021) &4096 D1066  ; RK_05 #2入壳机构步序1（铝壳定位）  // RK_05 #2入壳机构铝壳定位平台伸缩气缸伸出步（D1066.12）
; rung 11: #2入壳机构单步运行中2（电芯定位&入壳）
@LD D1063.15  ; RK_05 #2入壳机构单步（SW）
ANDNOT D1064.02  ; RK_05 #2入壳机构单步运行中2（电芯定位&入壳）
OR D1064.02  ; RK_05 #2入壳机构单步运行中2（电芯定位&入壳）
AND W1.00  ; 手动模式
ANDNOT 200.01  ; 紧急停止
ANDNOT 200.04  ; 报警清除
ANDNOT D1060.07  ; RK_05 #2入壳机构异常标志（总）
ANDNOT D1077.00  ; RK_05 #2入壳机构复位（M）
ANDNOT D1068.01  ; RK_05 #2入壳机构步进条件2（电芯定位&入壳）
OUT D1064.02  ; RK_05 #2入壳机构单步运行中2（电芯定位&入壳）
; rung 12
LD W1.00  ; 手动模式
ANDNOT 200.01  ; 紧急停止
ANDNOT 200.04  ; 报警清除
ANDNOT D1060.07  ; RK_05 #2入壳机构异常标志（总）
ANDNOT D1077.00  ; RK_05 #2入壳机构复位（M）
ANDNOT D1068.01  ; RK_05 #2入壳机构步进条件2（电芯定位&入壳）
OUT D1064.11  ; RK_05 #2入壳机构单步运行条件2（电芯定位&入壳）

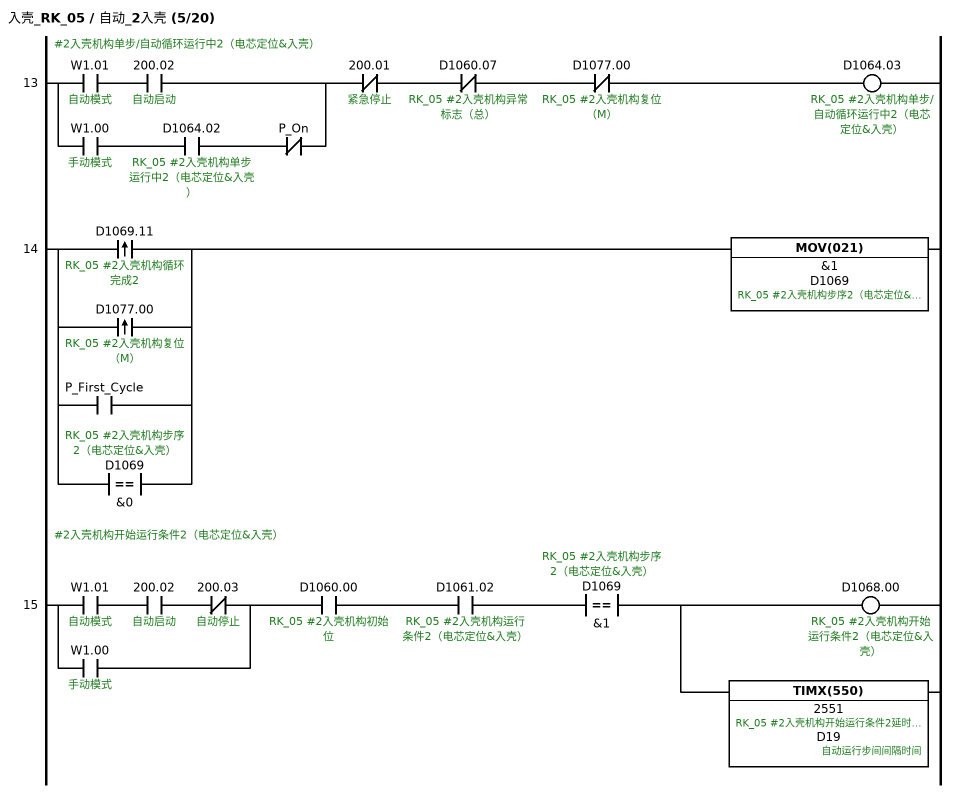
; rung 13: #2入壳机构单步/自动循环运行中2（电芯定位&入壳）
LD W1.01  ; 自动模式
AND 200.02  ; 自动启动
LD W1.00  ; 手动模式
AND D1064.02  ; RK_05 #2入壳机构单步运行中2（电芯定位&入壳）
ANDNOT P_On
ORLD
ANDNOT 200.01  ; 紧急停止
ANDNOT D1060.07  ; RK_05 #2入壳机构异常标志（总）
ANDNOT D1077.00  ; RK_05 #2入壳机构复位（M）
OUT D1064.03  ; RK_05 #2入壳机构单步/自动循环运行中2（电芯定位&入壳）
; rung 14
@LD D1069.11  ; RK_05 #2入壳机构循环完成2
@OR D1077.00  ; RK_05 #2入壳机构复位（M）
OR P_First_Cycle
OR=(300) D1069 &0  ; RK_05 #2入壳机构步序2（电芯定位&入壳）
MOV(021) &1 D1069  ; RK_05 #2入壳机构步序2（电芯定位&入壳）
; rung 15: #2入壳机构开始运行条件2（电芯定位&入壳）
LD W1.01  ; 自动模式
AND 200.02  ; 自动启动
ANDNOT 200.03  ; 自动停止
OR W1.00  ; 手动模式
AND D1060.00  ; RK_05 #2入壳机构初始位
AND D1061.02  ; RK_05 #2入壳机构运行条件2（电芯定位&入壳）
AND=(300) D1069 &1  ; RK_05 #2入壳机构步序2（电芯定位&入壳）
OUT D1068.00  ; RK_05 #2入壳机构开始运行条件2（电芯定位&入壳）
TIMX(550) 2551 D19  ; 自动运行步间间隔时间, RK_05 #2入壳机构开始运行条件2延时（电芯定位&入壳）

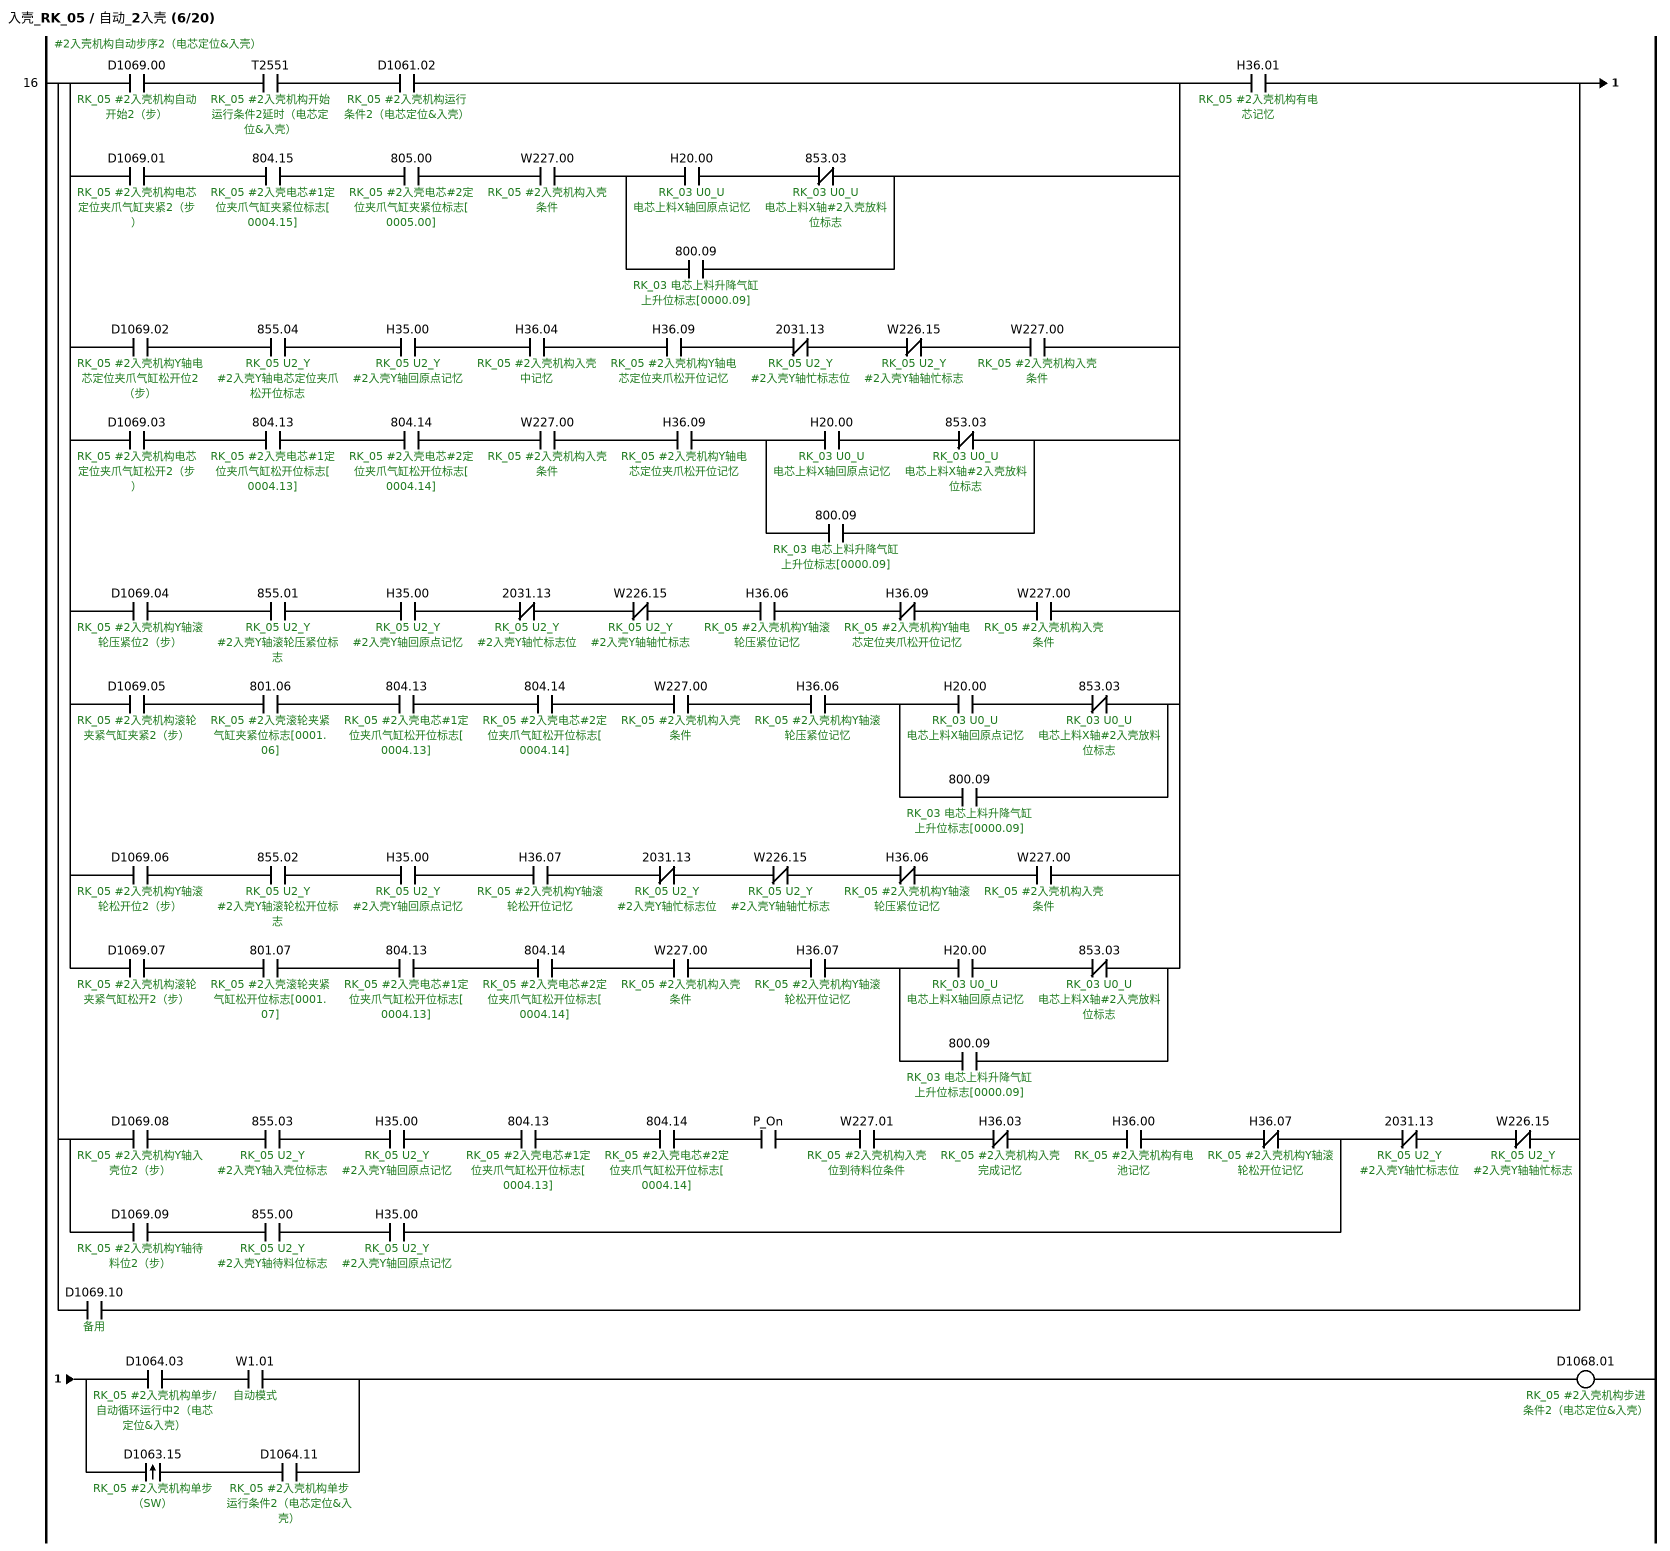
; rung 16: #2入壳机构自动步序2（电芯定位&入壳）
LD D1069.00  ; RK_05 #2入壳机构自动开始2（步）
AND T2551  ; RK_05 #2入壳机构开始运行条件2延时（电芯定位&入壳）
AND D1061.02  ; RK_05 #2入壳机构运行条件2（电芯定位&入壳）
LD D1069.01  ; RK_05 #2入壳机构电芯定位夹爪气缸夹紧2（步）
AND 804.15  ; RK_05 #2入壳电芯#1定位夹爪气缸夹紧位标志[0004.15]
AND 805.00  ; RK_05 #2入壳电芯#2定位夹爪气缸夹紧位标志[0005.00]
AND W227.00  ; RK_05 #2入壳机构入壳条件
LD H20.00  ; RK_03 U0_U 电芯上料X轴回原点记忆
ANDNOT 853.03  ; RK_03 U0_U 电芯上料X轴#2入壳放料位标志
OR 800.09  ; RK_03 电芯上料升降气缸上升位标志[0000.09]
ANDLD
ORLD
LD D1069.02  ; RK_05 #2入壳机构Y轴电芯定位夹爪气缸松开位2（步）
AND 855.04  ; RK_05 U2_Y #2入壳Y轴电芯定位夹爪松开位标志
AND H35.00  ; RK_05 U2_Y #2入壳Y轴回原点记忆
AND H36.04  ; RK_05 #2入壳机构入壳中记忆
AND H36.09  ; RK_05 #2入壳机构Y轴电芯定位夹爪松开位记忆
ANDNOT 2031.13  ; RK_05 U2_Y #2入壳Y轴忙标志位
ANDNOT W226.15  ; RK_05 U2_Y #2入壳Y轴轴忙标志
AND W227.00  ; RK_05 #2入壳机构入壳条件
ORLD
LD D1069.03  ; RK_05 #2入壳机构电芯定位夹爪气缸松开2（步）
AND 804.13  ; RK_05 #2入壳电芯#1定位夹爪气缸松开位标志[0004.13]
AND 804.14  ; RK_05 #2入壳电芯#2定位夹爪气缸松开位标志[0004.14]
AND W227.00  ; RK_05 #2入壳机构入壳条件
AND H36.09  ; RK_05 #2入壳机构Y轴电芯定位夹爪松开位记忆
LD H20.00  ; RK_03 U0_U 电芯上料X轴回原点记忆
ANDNOT 853.03  ; RK_03 U0_U 电芯上料X轴#2入壳放料位标志
OR 800.09  ; RK_03 电芯上料升降气缸上升位标志[0000.09]
ANDLD
ORLD
LD D1069.04  ; RK_05 #2入壳机构Y轴滚轮压紧位2（步）
AND 855.01  ; RK_05 U2_Y #2入壳Y轴滚轮压紧位标志
AND H35.00  ; RK_05 U2_Y #2入壳Y轴回原点记忆
ANDNOT 2031.13  ; RK_05 U2_Y #2入壳Y轴忙标志位
ANDNOT W226.15  ; RK_05 U2_Y #2入壳Y轴轴忙标志
AND H36.06  ; RK_05 #2入壳机构Y轴滚轮压紧位记忆
ANDNOT H36.09  ; RK_05 #2入壳机构Y轴电芯定位夹爪松开位记忆
AND W227.00  ; RK_05 #2入壳机构入壳条件
ORLD
LD D1069.05  ; RK_05 #2入壳机构滚轮夹紧气缸夹紧2（步）
AND 801.06  ; RK_05 #2入壳滚轮夹紧气缸夹紧位标志[0001.06]
AND 804.13  ; RK_05 #2入壳电芯#1定位夹爪气缸松开位标志[0004.13]
AND 804.14  ; RK_05 #2入壳电芯#2定位夹爪气缸松开位标志[0004.14]
AND W227.00  ; RK_05 #2入壳机构入壳条件
AND H36.06  ; RK_05 #2入壳机构Y轴滚轮压紧位记忆
LD H20.00  ; RK_03 U0_U 电芯上料X轴回原点记忆
ANDNOT 853.03  ; RK_03 U0_U 电芯上料X轴#2入壳放料位标志
OR 800.09  ; RK_03 电芯上料升降气缸上升位标志[0000.09]
ANDLD
ORLD
LD D1069.06  ; RK_05 #2入壳机构Y轴滚轮松开位2（步）
AND 855.02  ; RK_05 U2_Y #2入壳Y轴滚轮松开位标志
AND H35.00  ; RK_05 U2_Y #2入壳Y轴回原点记忆
AND H36.07  ; RK_05 #2入壳机构Y轴滚轮松开位记忆
ANDNOT 2031.13  ; RK_05 U2_Y #2入壳Y轴忙标志位
ANDNOT W226.15  ; RK_05 U2_Y #2入壳Y轴轴忙标志
ANDNOT H36.06  ; RK_05 #2入壳机构Y轴滚轮压紧位记忆
AND W227.00  ; RK_05 #2入壳机构入壳条件
ORLD
LD D1069.07  ; RK_05 #2入壳机构滚轮夹紧气缸松开2（步）
AND 801.07  ; RK_05 #2入壳滚轮夹紧气缸松开位标志[0001.07]
AND 804.13  ; RK_05 #2入壳电芯#1定位夹爪气缸松开位标志[0004.13]
AND 804.14  ; RK_05 #2入壳电芯#2定位夹爪气缸松开位标志[0004.14]
AND W227.00  ; RK_05 #2入壳机构入壳条件
AND H36.07  ; RK_05 #2入壳机构Y轴滚轮松开位记忆
LD H20.00  ; RK_03 U0_U 电芯上料X轴回原点记忆
ANDNOT 853.03  ; RK_03 U0_U 电芯上料X轴#2入壳放料位标志
OR 800.09  ; RK_03 电芯上料升降气缸上升位标志[0000.09]
ANDLD
ORLD
AND H36.01  ; RK_05 #2入壳机构有电芯记忆
LD D1069.08  ; RK_05 #2入壳机构Y轴入壳位2（步）
AND 855.03  ; RK_05 U2_Y #2入壳Y轴入壳位标志
AND H35.00  ; RK_05 U2_Y #2入壳Y轴回原点记忆
AND 804.13  ; RK_05 #2入壳电芯#1定位夹爪气缸松开位标志[0004.13]
AND 804.14  ; RK_05 #2入壳电芯#2定位夹爪气缸松开位标志[0004.14]
AND P_On  // 是否增加到入壳位后稳定延时？
AND W227.01  ; RK_05 #2入壳机构入壳位到待料位条件
ANDNOT H36.03  ; RK_05 #2入壳机构入壳完成记忆
AND H36.00  ; RK_05 #2入壳机构有电池记忆
ANDNOT H36.07  ; RK_05 #2入壳机构Y轴滚轮松开位记忆
LD D1069.09  ; RK_05 #2入壳机构Y轴待料位2（步）
AND 855.00  ; RK_05 U2_Y #2入壳Y轴待料位标志
AND H35.00  ; RK_05 U2_Y #2入壳Y轴回原点记忆
ORLD
ANDNOT 2031.13  ; RK_05 U2_Y #2入壳Y轴忙标志位
ANDNOT W226.15  ; RK_05 U2_Y #2入壳Y轴轴忙标志
ORLD
OR D1069.10  ; 备用
LD D1064.03  ; RK_05 #2入壳机构单步/自动循环运行中2（电芯定位&入壳）
AND W1.01  ; 自动模式
@LD D1063.15  ; RK_05 #2入壳机构单步（SW）
AND D1064.11  ; RK_05 #2入壳机构单步运行条件2（电芯定位&入壳）
ORLD
ANDLD
OUT D1068.01  ; RK_05 #2入壳机构步进条件2（电芯定位&入壳）

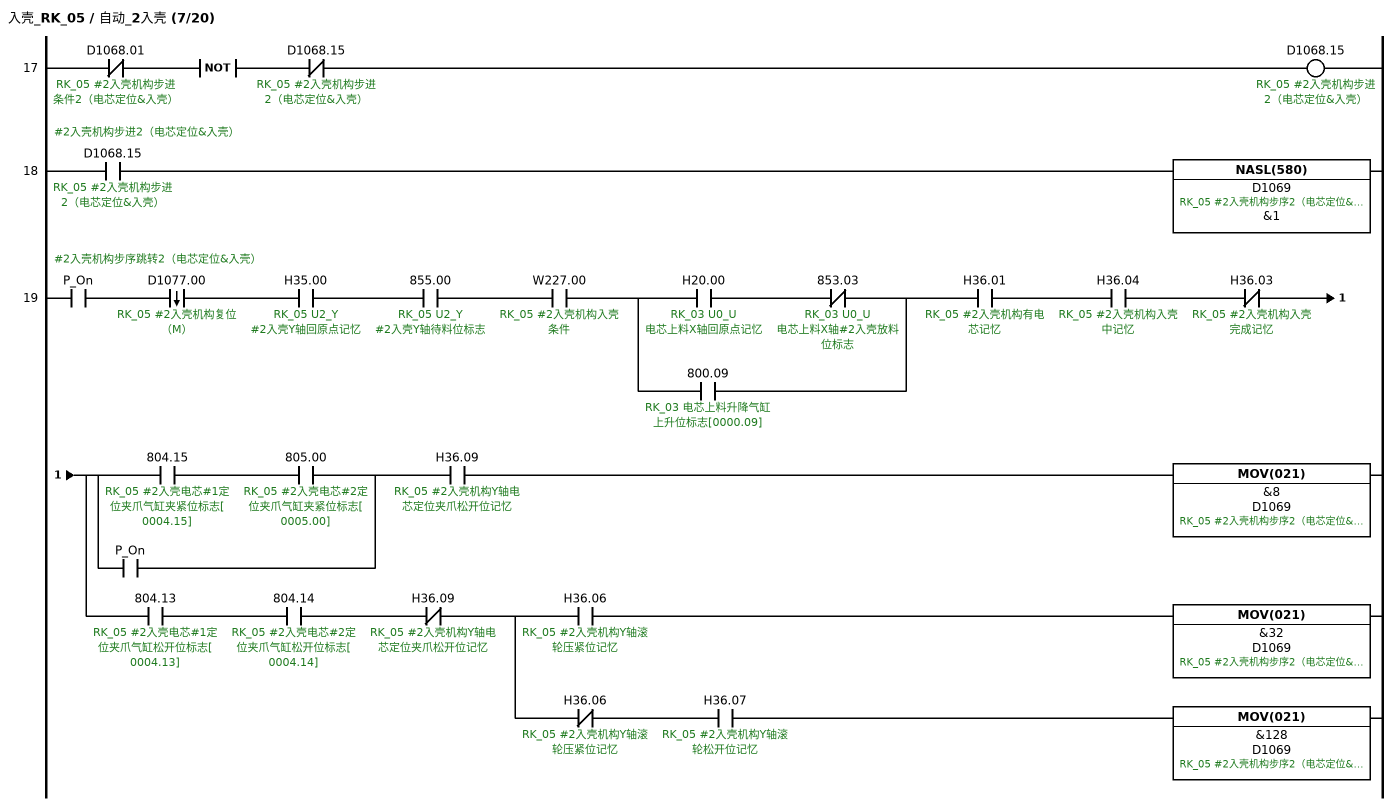
; rung 17
LDNOT D1068.01  ; RK_05 #2入壳机构步进条件2（电芯定位&入壳）
NOT(520)
ANDNOT D1068.15  ; RK_05 #2入壳机构步进2（电芯定位&入壳）
OUT D1068.15  ; RK_05 #2入壳机构步进2（电芯定位&入壳）
; rung 18: #2入壳机构步进2（电芯定位&入壳）
LD D1068.15  ; RK_05 #2入壳机构步进2（电芯定位&入壳）
NASL(580) D1069 &1  ; RK_05 #2入壳机构步序2（电芯定位&入壳）
; rung 19: #2入壳机构步序跳转2（电芯定位&入壳）
LD P_On
%AND D1077.00  ; RK_05 #2入壳机构复位（M）
AND H35.00  ; RK_05 U2_Y #2入壳Y轴回原点记忆
AND 855.00  ; RK_05 U2_Y #2入壳Y轴待料位标志
AND W227.00  ; RK_05 #2入壳机构入壳条件
LD H20.00  ; RK_03 U0_U 电芯上料X轴回原点记忆
ANDNOT 853.03  ; RK_03 U0_U 电芯上料X轴#2入壳放料位标志
OR 800.09  ; RK_03 电芯上料升降气缸上升位标志[0000.09]
ANDLD
AND H36.01  ; RK_05 #2入壳机构有电芯记忆
AND H36.04  ; RK_05 #2入壳机构入壳中记忆
ANDNOT H36.03  ; RK_05 #2入壳机构入壳完成记忆
OUT TR0
LD 804.15  ; RK_05 #2入壳电芯#1定位夹爪气缸夹紧位标志[0004.15]
AND 805.00  ; RK_05 #2入壳电芯#2定位夹爪气缸夹紧位标志[0005.00]
OR P_On
ANDLD
AND H36.09  ; RK_05 #2入壳机构Y轴电芯定位夹爪松开位记忆
MOV(021) &8 D1069  ; RK_05 #2入壳机构步序2（电芯定位&入壳）  // RK_05 #2入壳机构电芯定位夹爪气缸松开2步（D1069.03）
LD TR0
AND 804.13  ; RK_05 #2入壳电芯#1定位夹爪气缸松开位标志[0004.13]
AND 804.14  ; RK_05 #2入壳电芯#2定位夹爪气缸松开位标志[0004.14]
ANDNOT H36.09  ; RK_05 #2入壳机构Y轴电芯定位夹爪松开位记忆
OUT TR0
AND H36.06  ; RK_05 #2入壳机构Y轴滚轮压紧位记忆
MOV(021) &32 D1069  ; RK_05 #2入壳机构步序2（电芯定位&入壳）  // RK_05 #2入壳机构滚轮夹紧气缸夹紧2步（D1069.05）
LD TR0
ANDNOT H36.06  ; RK_05 #2入壳机构Y轴滚轮压紧位记忆
AND H36.07  ; RK_05 #2入壳机构Y轴滚轮松开位记忆
MOV(021) &128 D1069  ; RK_05 #2入壳机构步序2（电芯定位&入壳）  // RK_05 #2入壳机构滚轮夹紧气缸松开2步（D1069.08）

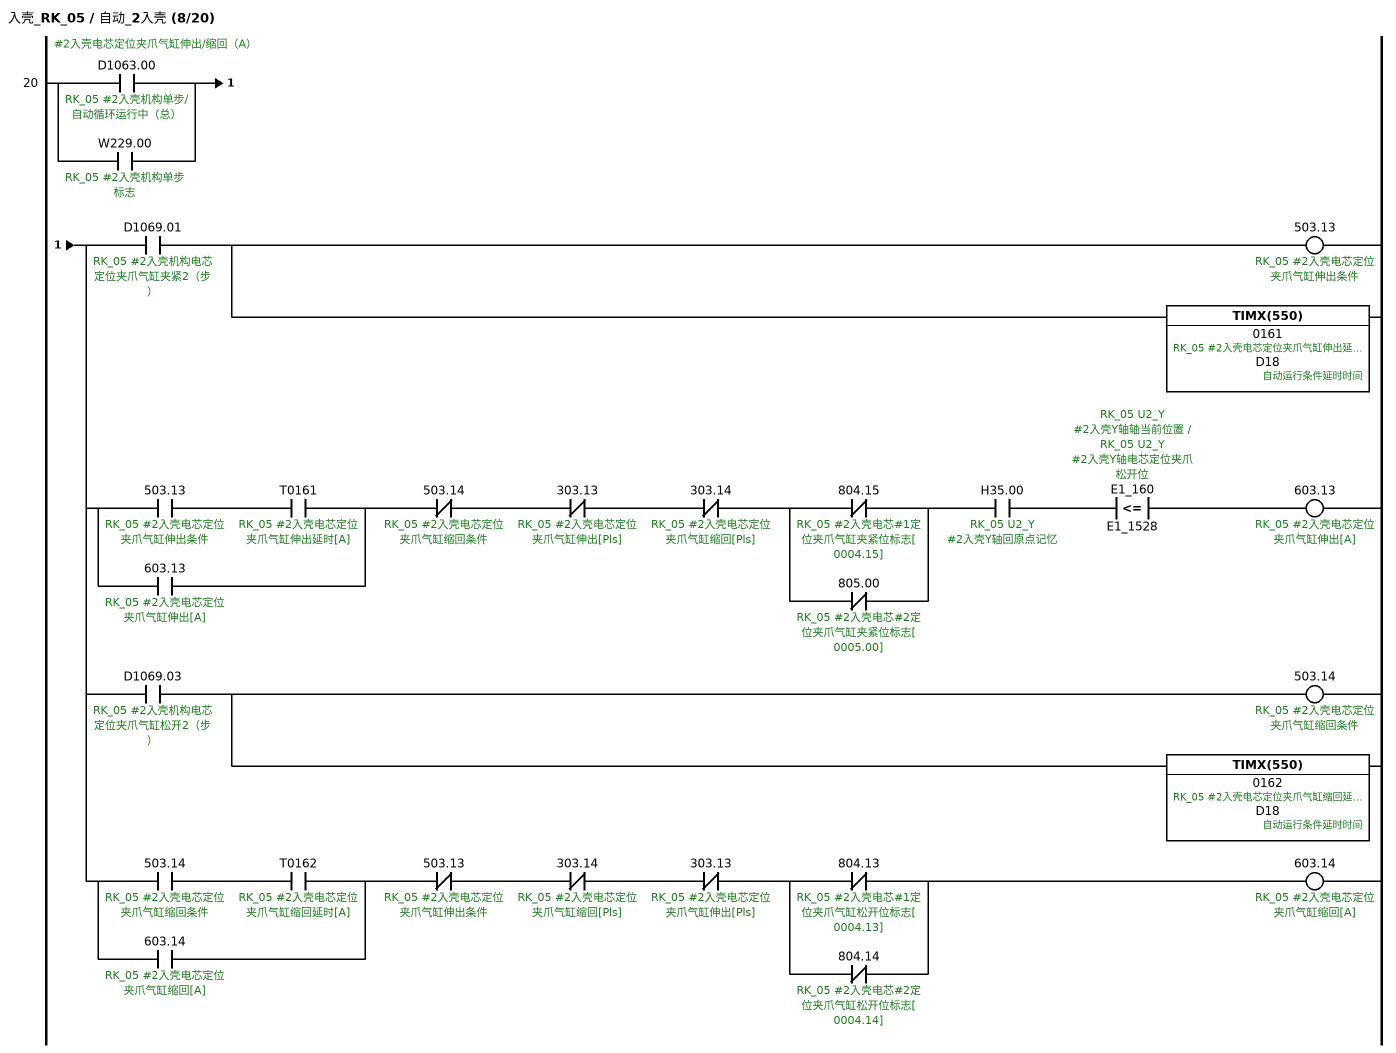
; rung 20: #2入壳电芯定位夹爪气缸伸出/缩回（A）
LD D1063.00  ; RK_05 #2入壳机构单步/自动循环运行中（总）
OR W229.00  ; RK_05 #2入壳机构单步标志
OUT TR0
AND D1069.01  ; RK_05 #2入壳机构电芯定位夹爪气缸夹紧2（步）
OUT 503.13  ; RK_05 #2入壳电芯定位夹爪气缸伸出条件
TIMX(550) 0161 D18  ; 自动运行条件延时时间, RK_05 #2入壳电芯定位夹爪气缸伸出延时[A]
LD TR0
LD 503.13  ; RK_05 #2入壳电芯定位夹爪气缸伸出条件
AND T0161  ; RK_05 #2入壳电芯定位夹爪气缸伸出延时[A]
OR 603.13  ; RK_05 #2入壳电芯定位夹爪气缸伸出[A]
ANDLD
ANDNOT 503.14  ; RK_05 #2入壳电芯定位夹爪气缸缩回条件
ANDNOT 303.13  ; RK_05 #2入壳电芯定位夹爪气缸伸出[Pls]
ANDNOT 303.14  ; RK_05 #2入壳电芯定位夹爪气缸缩回[Pls]
LDNOT 804.15  ; RK_05 #2入壳电芯#1定位夹爪气缸夹紧位标志[0004.15]
ORNOT 805.00  ; RK_05 #2入壳电芯#2定位夹爪气缸夹紧位标志[0005.00]
ANDLD
AND H35.00  ; RK_05 U2_Y #2入壳Y轴回原点记忆
AND<=SL(318) E1_160 E1_1528  ; RK_05 U2_Y #2入壳Y轴轴当前位置, RK_05 U2_Y #2入壳Y轴电芯定位夹爪松开位
OUT 603.13  ; RK_05 #2入壳电芯定位夹爪气缸伸出[A]
LD TR0
AND D1069.03  ; RK_05 #2入壳机构电芯定位夹爪气缸松开2（步）
OUT 503.14  ; RK_05 #2入壳电芯定位夹爪气缸缩回条件
TIMX(550) 0162 D18  ; 自动运行条件延时时间, RK_05 #2入壳电芯定位夹爪气缸缩回延时[A]
LD TR0
LD 503.14  ; RK_05 #2入壳电芯定位夹爪气缸缩回条件
AND T0162  ; RK_05 #2入壳电芯定位夹爪气缸缩回延时[A]
OR 603.14  ; RK_05 #2入壳电芯定位夹爪气缸缩回[A]
ANDLD
ANDNOT 503.13  ; RK_05 #2入壳电芯定位夹爪气缸伸出条件
ANDNOT 303.14  ; RK_05 #2入壳电芯定位夹爪气缸缩回[Pls]
ANDNOT 303.13  ; RK_05 #2入壳电芯定位夹爪气缸伸出[Pls]
LDNOT 804.13  ; RK_05 #2入壳电芯#1定位夹爪气缸松开位标志[0004.13]
ORNOT 804.14  ; RK_05 #2入壳电芯#2定位夹爪气缸松开位标志[0004.14]
ANDLD
OUT 603.14  ; RK_05 #2入壳电芯定位夹爪气缸缩回[A]

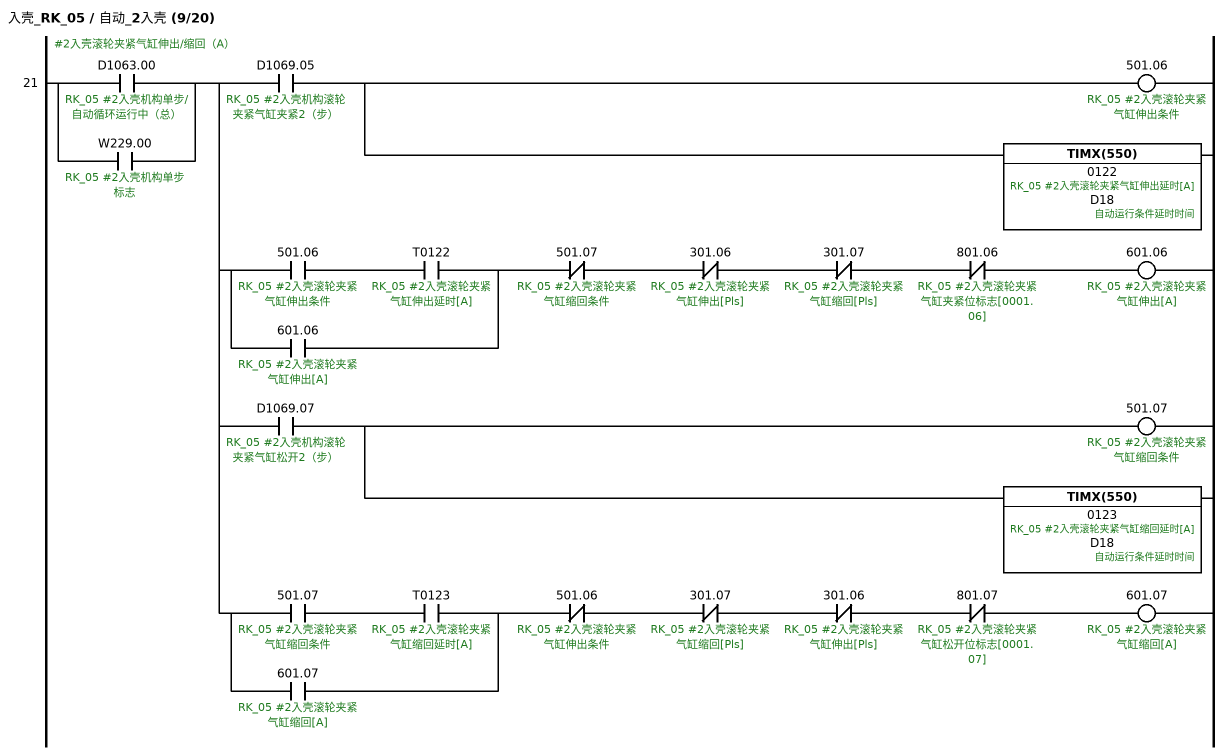
; rung 21: #2入壳滚轮夹紧气缸伸出/缩回（A）
LD D1063.00  ; RK_05 #2入壳机构单步/自动循环运行中（总）
OR W229.00  ; RK_05 #2入壳机构单步标志
OUT TR0
AND D1069.05  ; RK_05 #2入壳机构滚轮夹紧气缸夹紧2（步）
OUT 501.06  ; RK_05 #2入壳滚轮夹紧气缸伸出条件
TIMX(550) 0122 D18  ; 自动运行条件延时时间, RK_05 #2入壳滚轮夹紧气缸伸出延时[A]
LD TR0
LD 501.06  ; RK_05 #2入壳滚轮夹紧气缸伸出条件
AND T0122  ; RK_05 #2入壳滚轮夹紧气缸伸出延时[A]
OR 601.06  ; RK_05 #2入壳滚轮夹紧气缸伸出[A]
ANDLD
ANDNOT 501.07  ; RK_05 #2入壳滚轮夹紧气缸缩回条件
ANDNOT 301.06  ; RK_05 #2入壳滚轮夹紧气缸伸出[Pls]
ANDNOT 301.07  ; RK_05 #2入壳滚轮夹紧气缸缩回[Pls]
ANDNOT 801.06  ; RK_05 #2入壳滚轮夹紧气缸夹紧位标志[0001.06]
OUT 601.06  ; RK_05 #2入壳滚轮夹紧气缸伸出[A]
LD TR0
AND D1069.07  ; RK_05 #2入壳机构滚轮夹紧气缸松开2（步）
OUT 501.07  ; RK_05 #2入壳滚轮夹紧气缸缩回条件
TIMX(550) 0123 D18  ; 自动运行条件延时时间, RK_05 #2入壳滚轮夹紧气缸缩回延时[A]
LD TR0
LD 501.07  ; RK_05 #2入壳滚轮夹紧气缸缩回条件
AND T0123  ; RK_05 #2入壳滚轮夹紧气缸缩回延时[A]
OR 601.07  ; RK_05 #2入壳滚轮夹紧气缸缩回[A]
ANDLD
ANDNOT 501.06  ; RK_05 #2入壳滚轮夹紧气缸伸出条件
ANDNOT 301.07  ; RK_05 #2入壳滚轮夹紧气缸缩回[Pls]
ANDNOT 301.06  ; RK_05 #2入壳滚轮夹紧气缸伸出[Pls]
ANDNOT 801.07  ; RK_05 #2入壳滚轮夹紧气缸松开位标志[0001.07]
OUT 601.07  ; RK_05 #2入壳滚轮夹紧气缸缩回[A]

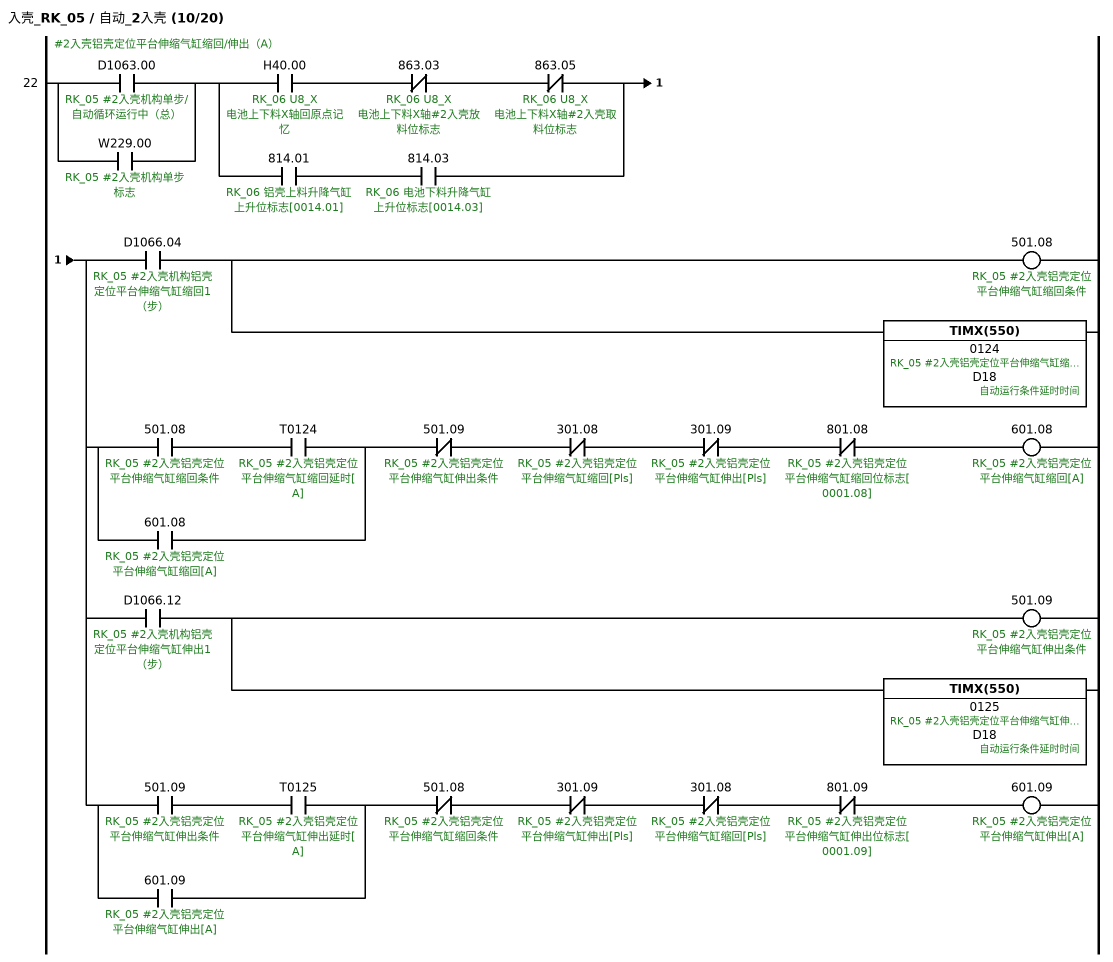
; rung 22: #2入壳铝壳定位平台伸缩气缸缩回/伸出（A）
LD D1063.00  ; RK_05 #2入壳机构单步/自动循环运行中（总）
OR W229.00  ; RK_05 #2入壳机构单步标志
LD H40.00  ; RK_06 U8_X 电池上下料X轴回原点记忆
ANDNOT 863.03  ; RK_06 U8_X 电池上下料X轴#2入壳放料位标志
ANDNOT 863.05  ; RK_06 U8_X 电池上下料X轴#2入壳取料位标志
LD 814.01  ; RK_06 铝壳上料升降气缸上升位标志[0014.01]
AND 814.03  ; RK_06 电池下料升降气缸上升位标志[0014.03]
ORLD
ANDLD
OUT TR0
AND D1066.04  ; RK_05 #2入壳机构铝壳定位平台伸缩气缸缩回1（步）
OUT 501.08  ; RK_05 #2入壳铝壳定位平台伸缩气缸缩回条件
TIMX(550) 0124 D18  ; 自动运行条件延时时间, RK_05 #2入壳铝壳定位平台伸缩气缸缩回延时[A]
LD TR0
LD 501.08  ; RK_05 #2入壳铝壳定位平台伸缩气缸缩回条件
AND T0124  ; RK_05 #2入壳铝壳定位平台伸缩气缸缩回延时[A]
OR 601.08  ; RK_05 #2入壳铝壳定位平台伸缩气缸缩回[A]
ANDLD
ANDNOT 501.09  ; RK_05 #2入壳铝壳定位平台伸缩气缸伸出条件
ANDNOT 301.08  ; RK_05 #2入壳铝壳定位平台伸缩气缸缩回[Pls]
ANDNOT 301.09  ; RK_05 #2入壳铝壳定位平台伸缩气缸伸出[Pls]
ANDNOT 801.08  ; RK_05 #2入壳铝壳定位平台伸缩气缸缩回位标志[0001.08]
OUT 601.08  ; RK_05 #2入壳铝壳定位平台伸缩气缸缩回[A]
LD TR0
AND D1066.12  ; RK_05 #2入壳机构铝壳定位平台伸缩气缸伸出1（步）
OUT 501.09  ; RK_05 #2入壳铝壳定位平台伸缩气缸伸出条件
TIMX(550) 0125 D18  ; 自动运行条件延时时间, RK_05 #2入壳铝壳定位平台伸缩气缸伸出延时[A]
LD TR0
LD 501.09  ; RK_05 #2入壳铝壳定位平台伸缩气缸伸出条件
AND T0125  ; RK_05 #2入壳铝壳定位平台伸缩气缸伸出延时[A]
OR 601.09  ; RK_05 #2入壳铝壳定位平台伸缩气缸伸出[A]
ANDLD
ANDNOT 501.08  ; RK_05 #2入壳铝壳定位平台伸缩气缸缩回条件
ANDNOT 301.09  ; RK_05 #2入壳铝壳定位平台伸缩气缸伸出[Pls]
ANDNOT 301.08  ; RK_05 #2入壳铝壳定位平台伸缩气缸缩回[Pls]
ANDNOT 801.09  ; RK_05 #2入壳铝壳定位平台伸缩气缸伸出位标志[0001.09]
OUT 601.09  ; RK_05 #2入壳铝壳定位平台伸缩气缸伸出[A]

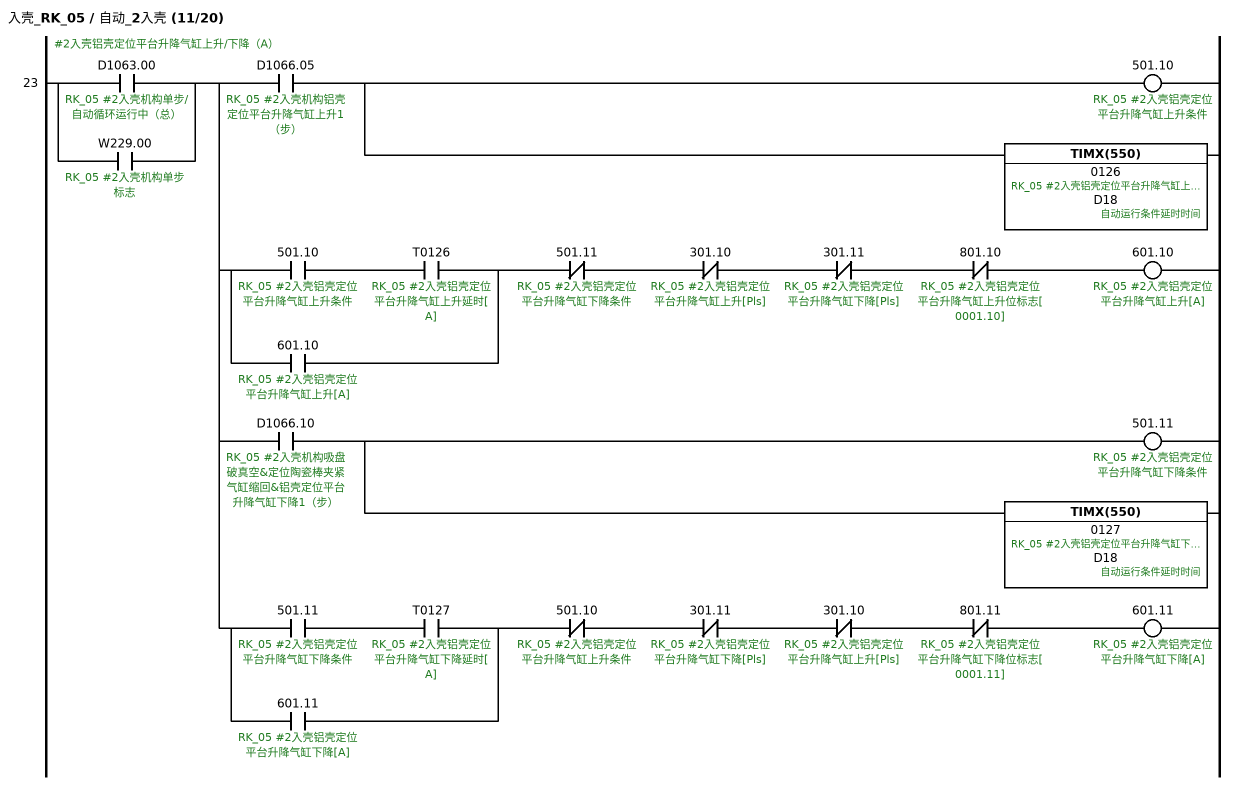
; rung 23: #2入壳铝壳定位平台升降气缸上升/下降（A）
LD D1063.00  ; RK_05 #2入壳机构单步/自动循环运行中（总）
OR W229.00  ; RK_05 #2入壳机构单步标志
OUT TR0
AND D1066.05  ; RK_05 #2入壳机构铝壳定位平台升降气缸上升1（步）
OUT 501.10  ; RK_05 #2入壳铝壳定位平台升降气缸上升条件
TIMX(550) 0126 D18  ; 自动运行条件延时时间, RK_05 #2入壳铝壳定位平台升降气缸上升延时[A]
LD TR0
LD 501.10  ; RK_05 #2入壳铝壳定位平台升降气缸上升条件
AND T0126  ; RK_05 #2入壳铝壳定位平台升降气缸上升延时[A]
OR 601.10  ; RK_05 #2入壳铝壳定位平台升降气缸上升[A]
ANDLD
ANDNOT 501.11  ; RK_05 #2入壳铝壳定位平台升降气缸下降条件
ANDNOT 301.10  ; RK_05 #2入壳铝壳定位平台升降气缸上升[Pls]
ANDNOT 301.11  ; RK_05 #2入壳铝壳定位平台升降气缸下降[Pls]
ANDNOT 801.10  ; RK_05 #2入壳铝壳定位平台升降气缸上升位标志[0001.10]
OUT 601.10  ; RK_05 #2入壳铝壳定位平台升降气缸上升[A]
LD TR0
AND D1066.10  ; RK_05 #2入壳机构吸盘破真空&定位陶瓷棒夹紧气缸缩回&铝壳定位平台升降气缸下降1（步）
OUT 501.11  ; RK_05 #2入壳铝壳定位平台升降气缸下降条件
TIMX(550) 0127 D18  ; 自动运行条件延时时间, RK_05 #2入壳铝壳定位平台升降气缸下降延时[A]
LD TR0
LD 501.11  ; RK_05 #2入壳铝壳定位平台升降气缸下降条件
AND T0127  ; RK_05 #2入壳铝壳定位平台升降气缸下降延时[A]
OR 601.11  ; RK_05 #2入壳铝壳定位平台升降气缸下降[A]
ANDLD
ANDNOT 501.10  ; RK_05 #2入壳铝壳定位平台升降气缸上升条件
ANDNOT 301.11  ; RK_05 #2入壳铝壳定位平台升降气缸下降[Pls]
ANDNOT 301.10  ; RK_05 #2入壳铝壳定位平台升降气缸上升[Pls]
ANDNOT 801.11  ; RK_05 #2入壳铝壳定位平台升降气缸下降位标志[0001.11]
OUT 601.11  ; RK_05 #2入壳铝壳定位平台升降气缸下降[A]

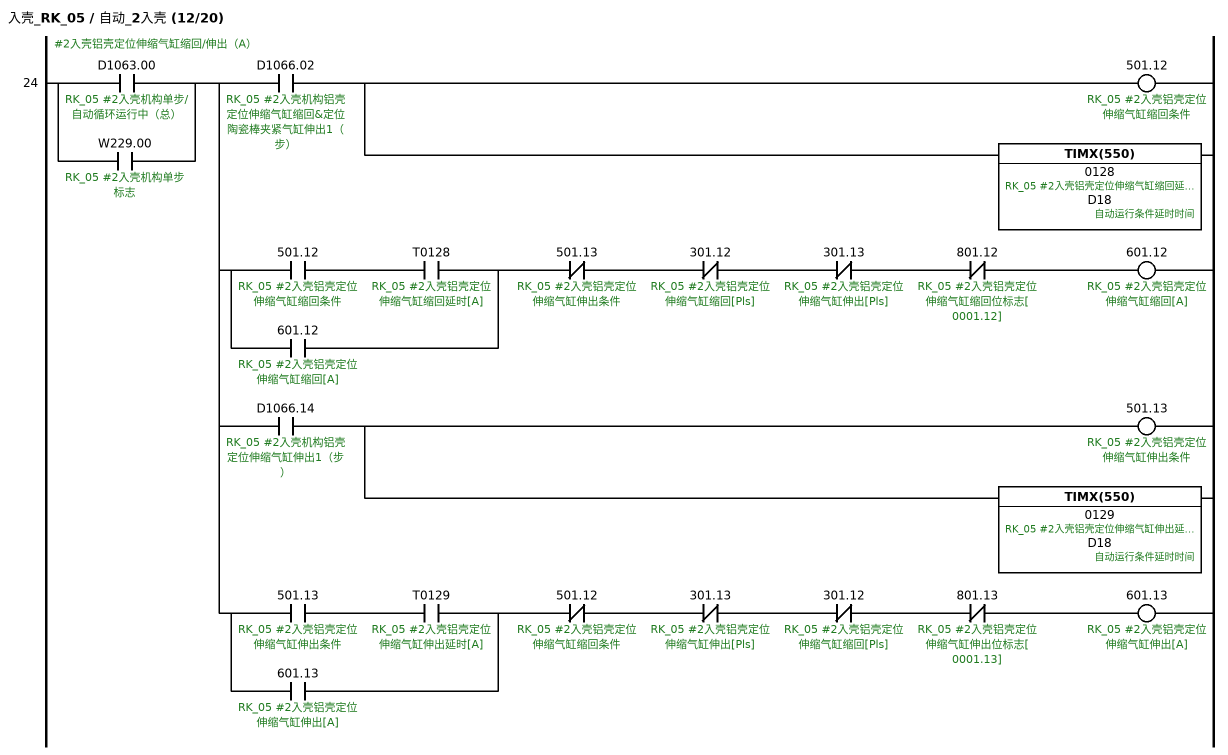
; rung 24: #2入壳铝壳定位伸缩气缸缩回/伸出（A）
LD D1063.00  ; RK_05 #2入壳机构单步/自动循环运行中（总）
OR W229.00  ; RK_05 #2入壳机构单步标志
OUT TR0
AND D1066.02  ; RK_05 #2入壳机构铝壳定位伸缩气缸缩回&定位陶瓷棒夹紧气缸伸出1（步）
OUT 501.12  ; RK_05 #2入壳铝壳定位伸缩气缸缩回条件
TIMX(550) 0128 D18  ; 自动运行条件延时时间, RK_05 #2入壳铝壳定位伸缩气缸缩回延时[A]
LD TR0
LD 501.12  ; RK_05 #2入壳铝壳定位伸缩气缸缩回条件
AND T0128  ; RK_05 #2入壳铝壳定位伸缩气缸缩回延时[A]
OR 601.12  ; RK_05 #2入壳铝壳定位伸缩气缸缩回[A]
ANDLD
ANDNOT 501.13  ; RK_05 #2入壳铝壳定位伸缩气缸伸出条件
ANDNOT 301.12  ; RK_05 #2入壳铝壳定位伸缩气缸缩回[Pls]
ANDNOT 301.13  ; RK_05 #2入壳铝壳定位伸缩气缸伸出[Pls]
ANDNOT 801.12  ; RK_05 #2入壳铝壳定位伸缩气缸缩回位标志[0001.12]
OUT 601.12  ; RK_05 #2入壳铝壳定位伸缩气缸缩回[A]
LD TR0
AND D1066.14  ; RK_05 #2入壳机构铝壳定位伸缩气缸伸出1（步）
OUT 501.13  ; RK_05 #2入壳铝壳定位伸缩气缸伸出条件
TIMX(550) 0129 D18  ; 自动运行条件延时时间, RK_05 #2入壳铝壳定位伸缩气缸伸出延时[A]
LD TR0
LD 501.13  ; RK_05 #2入壳铝壳定位伸缩气缸伸出条件
AND T0129  ; RK_05 #2入壳铝壳定位伸缩气缸伸出延时[A]
OR 601.13  ; RK_05 #2入壳铝壳定位伸缩气缸伸出[A]
ANDLD
ANDNOT 501.12  ; RK_05 #2入壳铝壳定位伸缩气缸缩回条件
ANDNOT 301.13  ; RK_05 #2入壳铝壳定位伸缩气缸伸出[Pls]
ANDNOT 301.12  ; RK_05 #2入壳铝壳定位伸缩气缸缩回[Pls]
ANDNOT 801.13  ; RK_05 #2入壳铝壳定位伸缩气缸伸出位标志[0001.13]
OUT 601.13  ; RK_05 #2入壳铝壳定位伸缩气缸伸出[A]

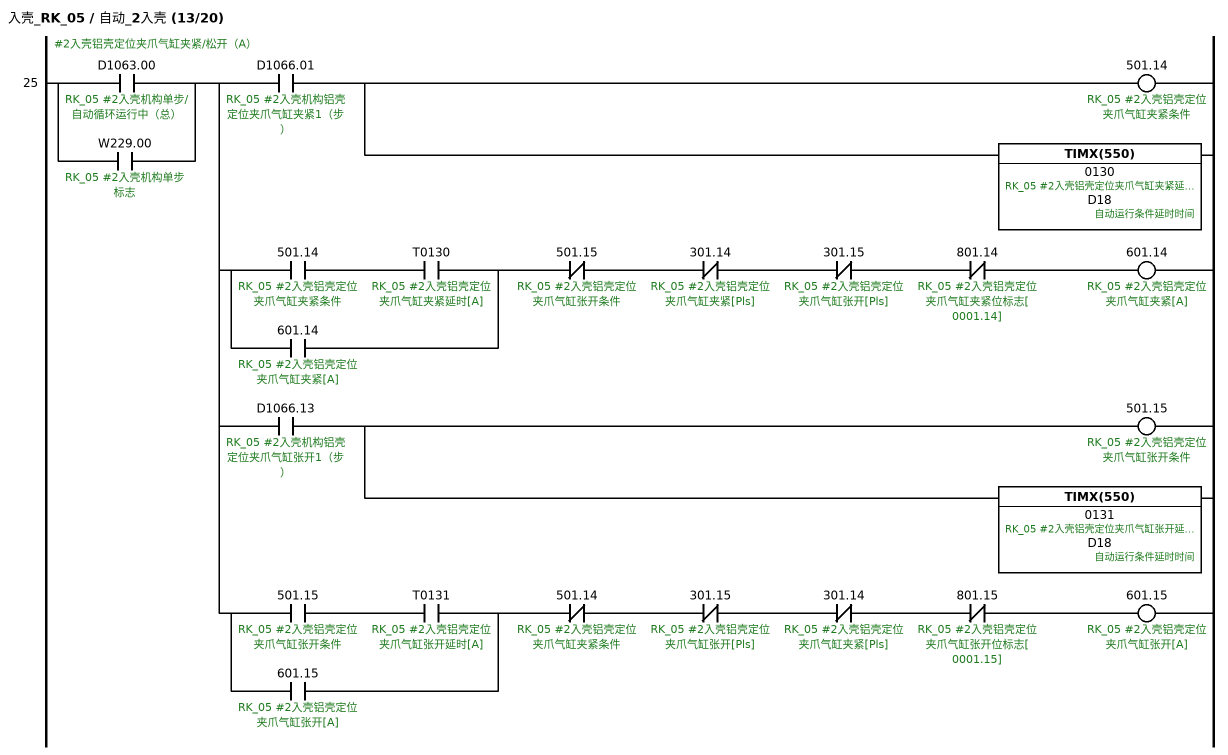
; rung 25: #2入壳铝壳定位夹爪气缸夹紧/松开（A）
LD D1063.00  ; RK_05 #2入壳机构单步/自动循环运行中（总）
OR W229.00  ; RK_05 #2入壳机构单步标志
OUT TR0
AND D1066.01  ; RK_05 #2入壳机构铝壳定位夹爪气缸夹紧1（步）
OUT 501.14  ; RK_05 #2入壳铝壳定位夹爪气缸夹紧条件
TIMX(550) 0130 D18  ; 自动运行条件延时时间, RK_05 #2入壳铝壳定位夹爪气缸夹紧延时[A]
LD TR0
LD 501.14  ; RK_05 #2入壳铝壳定位夹爪气缸夹紧条件
AND T0130  ; RK_05 #2入壳铝壳定位夹爪气缸夹紧延时[A]
OR 601.14  ; RK_05 #2入壳铝壳定位夹爪气缸夹紧[A]
ANDLD
ANDNOT 501.15  ; RK_05 #2入壳铝壳定位夹爪气缸张开条件
ANDNOT 301.14  ; RK_05 #2入壳铝壳定位夹爪气缸夹紧[Pls]
ANDNOT 301.15  ; RK_05 #2入壳铝壳定位夹爪气缸张开[Pls]
ANDNOT 801.14  ; RK_05 #2入壳铝壳定位夹爪气缸夹紧位标志[0001.14]
OUT 601.14  ; RK_05 #2入壳铝壳定位夹爪气缸夹紧[A]
LD TR0
AND D1066.13  ; RK_05 #2入壳机构铝壳定位夹爪气缸张开1（步）
OUT 501.15  ; RK_05 #2入壳铝壳定位夹爪气缸张开条件
TIMX(550) 0131 D18  ; 自动运行条件延时时间, RK_05 #2入壳铝壳定位夹爪气缸张开延时[A]
LD TR0
LD 501.15  ; RK_05 #2入壳铝壳定位夹爪气缸张开条件
AND T0131  ; RK_05 #2入壳铝壳定位夹爪气缸张开延时[A]
OR 601.15  ; RK_05 #2入壳铝壳定位夹爪气缸张开[A]
ANDLD
ANDNOT 501.14  ; RK_05 #2入壳铝壳定位夹爪气缸夹紧条件
ANDNOT 301.15  ; RK_05 #2入壳铝壳定位夹爪气缸张开[Pls]
ANDNOT 301.14  ; RK_05 #2入壳铝壳定位夹爪气缸夹紧[Pls]
ANDNOT 801.15  ; RK_05 #2入壳铝壳定位夹爪气缸张开位标志[0001.15]
OUT 601.15  ; RK_05 #2入壳铝壳定位夹爪气缸张开[A]

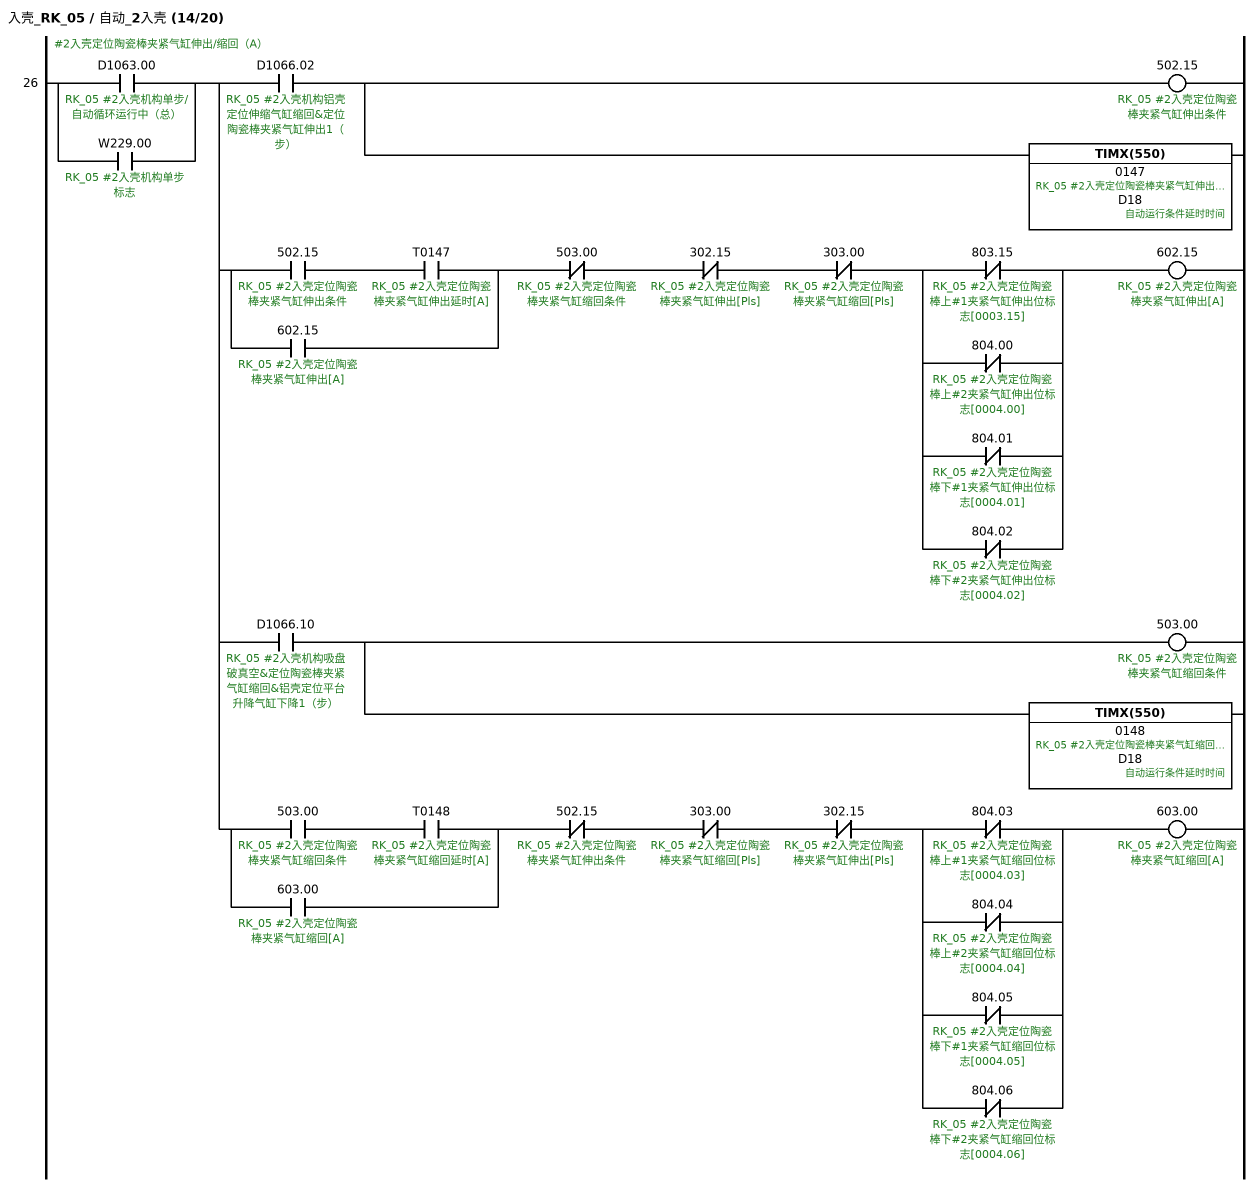
; rung 26: #2入壳定位陶瓷棒夹紧气缸伸出/缩回（A）
LD D1063.00  ; RK_05 #2入壳机构单步/自动循环运行中（总）
OR W229.00  ; RK_05 #2入壳机构单步标志
OUT TR0
AND D1066.02  ; RK_05 #2入壳机构铝壳定位伸缩气缸缩回&定位陶瓷棒夹紧气缸伸出1（步）
OUT 502.15  ; RK_05 #2入壳定位陶瓷棒夹紧气缸伸出条件
TIMX(550) 0147 D18  ; 自动运行条件延时时间, RK_05 #2入壳定位陶瓷棒夹紧气缸伸出延时[A]
LD TR0
LD 502.15  ; RK_05 #2入壳定位陶瓷棒夹紧气缸伸出条件
AND T0147  ; RK_05 #2入壳定位陶瓷棒夹紧气缸伸出延时[A]
OR 602.15  ; RK_05 #2入壳定位陶瓷棒夹紧气缸伸出[A]
ANDLD
ANDNOT 503.00  ; RK_05 #2入壳定位陶瓷棒夹紧气缸缩回条件
ANDNOT 302.15  ; RK_05 #2入壳定位陶瓷棒夹紧气缸伸出[Pls]
ANDNOT 303.00  ; RK_05 #2入壳定位陶瓷棒夹紧气缸缩回[Pls]
LDNOT 803.15  ; RK_05 #2入壳定位陶瓷棒上#1夹紧气缸伸出位标志[0003.15]
ORNOT 804.00  ; RK_05 #2入壳定位陶瓷棒上#2夹紧气缸伸出位标志[0004.00]
ORNOT 804.01  ; RK_05 #2入壳定位陶瓷棒下#1夹紧气缸伸出位标志[0004.01]
ORNOT 804.02  ; RK_05 #2入壳定位陶瓷棒下#2夹紧气缸伸出位标志[0004.02]
ANDLD
OUT 602.15  ; RK_05 #2入壳定位陶瓷棒夹紧气缸伸出[A]
LD TR0
AND D1066.10  ; RK_05 #2入壳机构吸盘破真空&定位陶瓷棒夹紧气缸缩回&铝壳定位平台升降气缸下降1（步）
OUT 503.00  ; RK_05 #2入壳定位陶瓷棒夹紧气缸缩回条件
TIMX(550) 0148 D18  ; 自动运行条件延时时间, RK_05 #2入壳定位陶瓷棒夹紧气缸缩回延时[A]
LD TR0
LD 503.00  ; RK_05 #2入壳定位陶瓷棒夹紧气缸缩回条件
AND T0148  ; RK_05 #2入壳定位陶瓷棒夹紧气缸缩回延时[A]
OR 603.00  ; RK_05 #2入壳定位陶瓷棒夹紧气缸缩回[A]
ANDLD
ANDNOT 502.15  ; RK_05 #2入壳定位陶瓷棒夹紧气缸伸出条件
ANDNOT 303.00  ; RK_05 #2入壳定位陶瓷棒夹紧气缸缩回[Pls]
ANDNOT 302.15  ; RK_05 #2入壳定位陶瓷棒夹紧气缸伸出[Pls]
LDNOT 804.03  ; RK_05 #2入壳定位陶瓷棒上#1夹紧气缸缩回位标志[0004.03]
ORNOT 804.04  ; RK_05 #2入壳定位陶瓷棒上#2夹紧气缸缩回位标志[0004.04]
ORNOT 804.05  ; RK_05 #2入壳定位陶瓷棒下#1夹紧气缸缩回位标志[0004.05]
ORNOT 804.06  ; RK_05 #2入壳定位陶瓷棒下#2夹紧气缸缩回位标志[0004.06]
ANDLD
OUT 603.00  ; RK_05 #2入壳定位陶瓷棒夹紧气缸缩回[A]

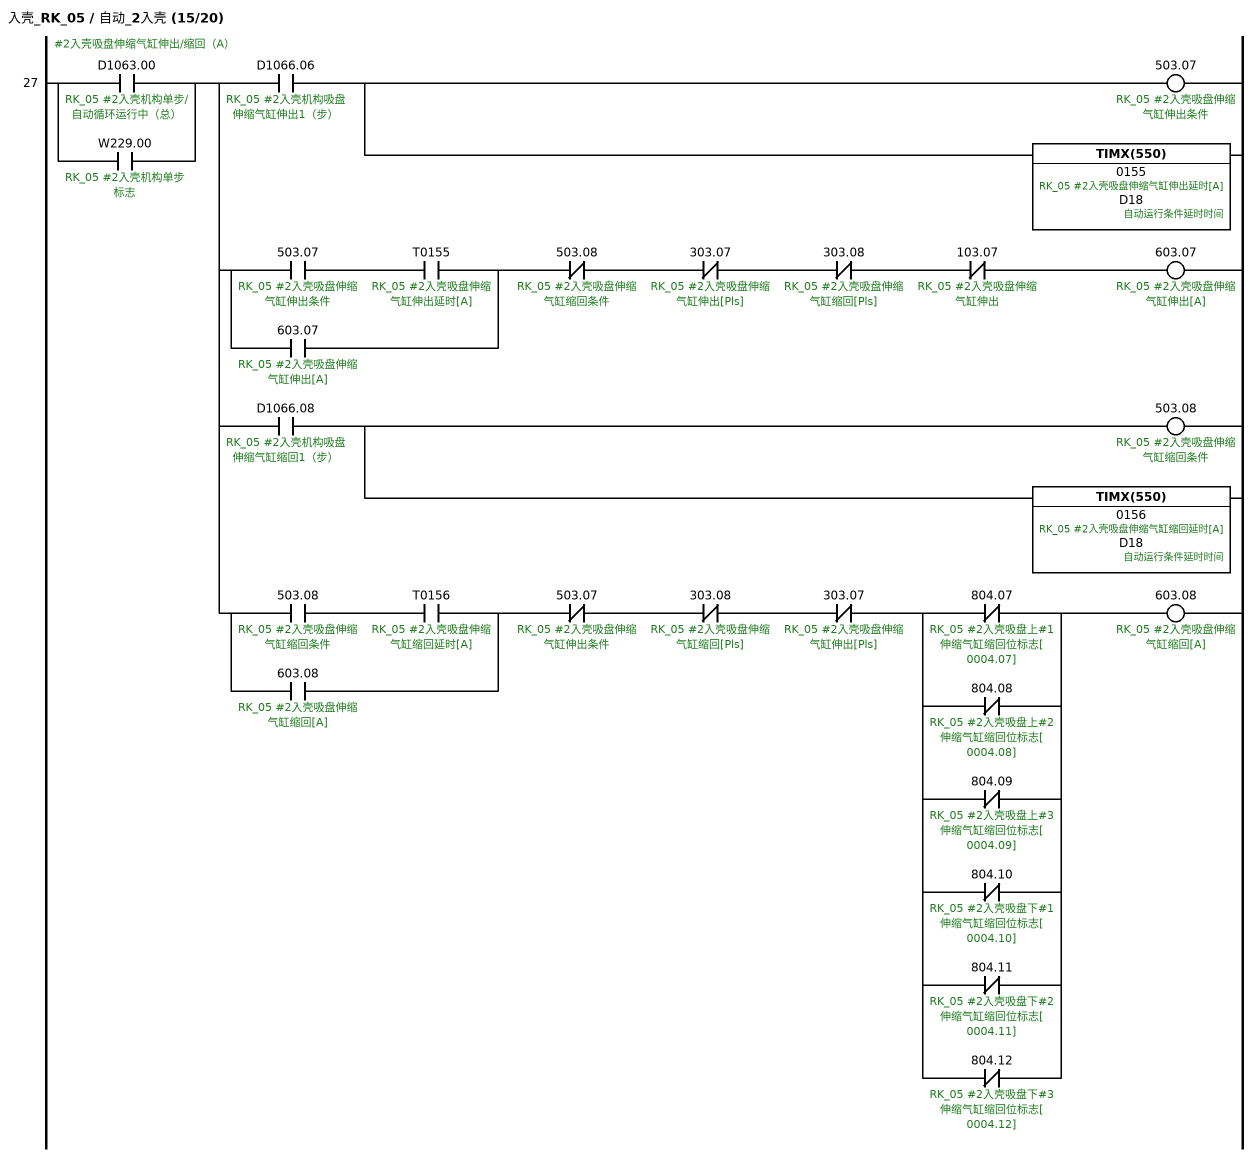
; rung 27: #2入壳吸盘伸缩气缸伸出/缩回（A）
LD D1063.00  ; RK_05 #2入壳机构单步/自动循环运行中（总）
OR W229.00  ; RK_05 #2入壳机构单步标志
OUT TR0
AND D1066.06  ; RK_05 #2入壳机构吸盘伸缩气缸伸出1（步）
OUT 503.07  ; RK_05 #2入壳吸盘伸缩气缸伸出条件
TIMX(550) 0155 D18  ; 自动运行条件延时时间, RK_05 #2入壳吸盘伸缩气缸伸出延时[A]
LD TR0
LD 503.07  ; RK_05 #2入壳吸盘伸缩气缸伸出条件
AND T0155  ; RK_05 #2入壳吸盘伸缩气缸伸出延时[A]
OR 603.07  ; RK_05 #2入壳吸盘伸缩气缸伸出[A]
ANDLD
ANDNOT 503.08  ; RK_05 #2入壳吸盘伸缩气缸缩回条件
ANDNOT 303.07  ; RK_05 #2入壳吸盘伸缩气缸伸出[Pls]
ANDNOT 303.08  ; RK_05 #2入壳吸盘伸缩气缸缩回[Pls]
ANDNOT 103.07  ; RK_05 #2入壳吸盘伸缩气缸伸出
OUT 603.07  ; RK_05 #2入壳吸盘伸缩气缸伸出[A]
LD TR0
AND D1066.08  ; RK_05 #2入壳机构吸盘伸缩气缸缩回1（步）
OUT 503.08  ; RK_05 #2入壳吸盘伸缩气缸缩回条件
TIMX(550) 0156 D18  ; 自动运行条件延时时间, RK_05 #2入壳吸盘伸缩气缸缩回延时[A]
LD TR0
LD 503.08  ; RK_05 #2入壳吸盘伸缩气缸缩回条件
AND T0156  ; RK_05 #2入壳吸盘伸缩气缸缩回延时[A]
OR 603.08  ; RK_05 #2入壳吸盘伸缩气缸缩回[A]
ANDLD
ANDNOT 503.07  ; RK_05 #2入壳吸盘伸缩气缸伸出条件
ANDNOT 303.08  ; RK_05 #2入壳吸盘伸缩气缸缩回[Pls]
ANDNOT 303.07  ; RK_05 #2入壳吸盘伸缩气缸伸出[Pls]
LDNOT 804.07  ; RK_05 #2入壳吸盘上#1伸缩气缸缩回位标志[0004.07]
ORNOT 804.08  ; RK_05 #2入壳吸盘上#2伸缩气缸缩回位标志[0004.08]
ORNOT 804.09  ; RK_05 #2入壳吸盘上#3伸缩气缸缩回位标志[0004.09]
ORNOT 804.10  ; RK_05 #2入壳吸盘下#1伸缩气缸缩回位标志[0004.10]
ORNOT 804.11  ; RK_05 #2入壳吸盘下#2伸缩气缸缩回位标志[0004.11]
ORNOT 804.12  ; RK_05 #2入壳吸盘下#3伸缩气缸缩回位标志[0004.12]
ANDLD
OUT 603.08  ; RK_05 #2入壳吸盘伸缩气缸缩回[A]

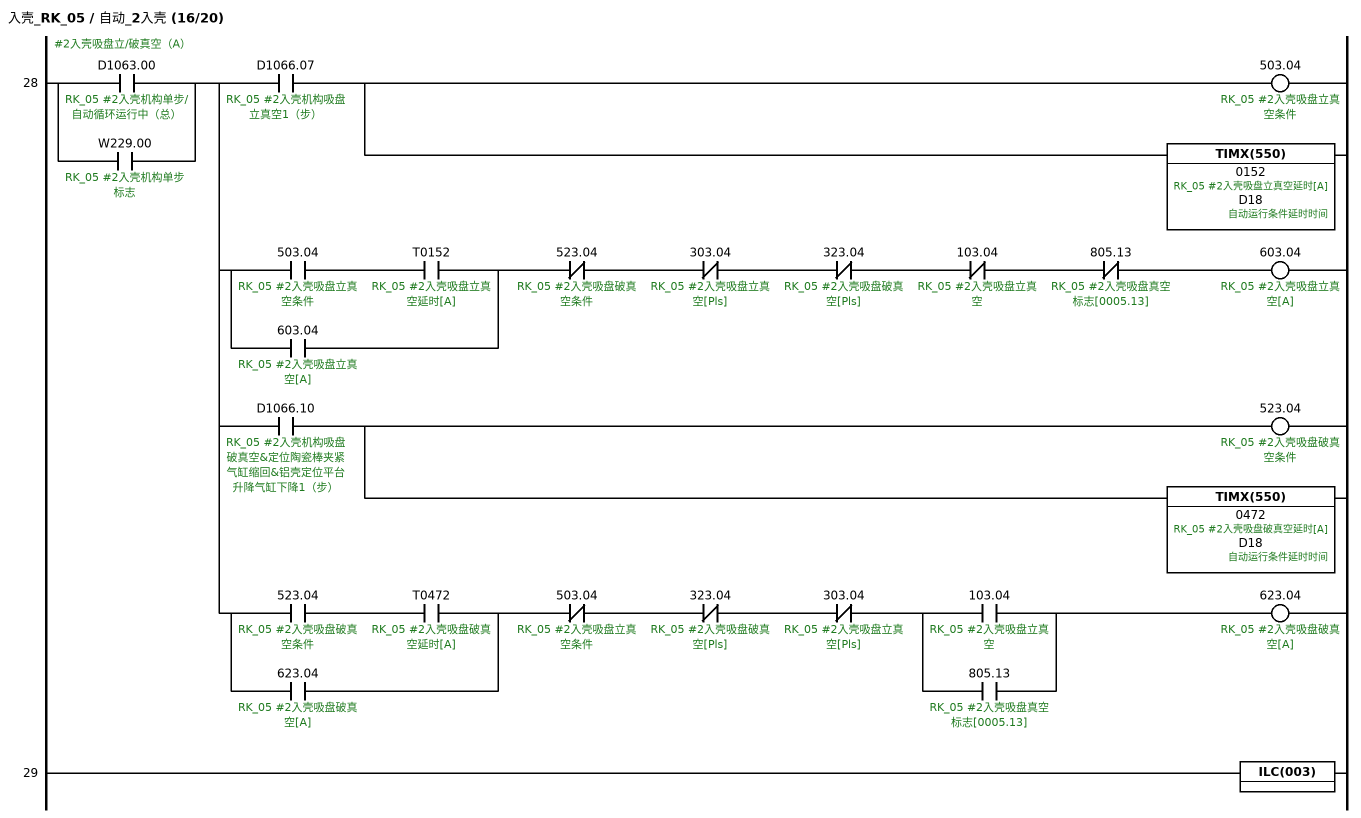
; rung 28: #2入壳吸盘立/破真空（A）
LD D1063.00  ; RK_05 #2入壳机构单步/自动循环运行中（总）
OR W229.00  ; RK_05 #2入壳机构单步标志
OUT TR0
AND D1066.07  ; RK_05 #2入壳机构吸盘立真空1（步）
OUT 503.04  ; RK_05 #2入壳吸盘立真空条件
TIMX(550) 0152 D18  ; 自动运行条件延时时间, RK_05 #2入壳吸盘立真空延时[A]
LD TR0
LD 503.04  ; RK_05 #2入壳吸盘立真空条件
AND T0152  ; RK_05 #2入壳吸盘立真空延时[A]
OR 603.04  ; RK_05 #2入壳吸盘立真空[A]
ANDLD
ANDNOT 523.04  ; RK_05 #2入壳吸盘破真空条件
ANDNOT 303.04  ; RK_05 #2入壳吸盘立真空[Pls]
ANDNOT 323.04  ; RK_05 #2入壳吸盘破真空[Pls]
ANDNOT 103.04  ; RK_05 #2入壳吸盘立真空
ANDNOT 805.13  ; RK_05 #2入壳吸盘真空标志[0005.13]
OUT 603.04  ; RK_05 #2入壳吸盘立真空[A]
LD TR0
AND D1066.10  ; RK_05 #2入壳机构吸盘破真空&定位陶瓷棒夹紧气缸缩回&铝壳定位平台升降气缸下降1（步）
OUT 523.04  ; RK_05 #2入壳吸盘破真空条件
TIMX(550) 0472 D18  ; 自动运行条件延时时间, RK_05 #2入壳吸盘破真空延时[A]
LD TR0
LD 523.04  ; RK_05 #2入壳吸盘破真空条件
AND T0472  ; RK_05 #2入壳吸盘破真空延时[A]
OR 623.04  ; RK_05 #2入壳吸盘破真空[A]
ANDLD
ANDNOT 503.04  ; RK_05 #2入壳吸盘立真空条件
ANDNOT 323.04  ; RK_05 #2入壳吸盘破真空[Pls]
ANDNOT 303.04  ; RK_05 #2入壳吸盘立真空[Pls]
LD 103.04  ; RK_05 #2入壳吸盘立真空
OR 805.13  ; RK_05 #2入壳吸盘真空标志[0005.13]
ANDLD
OUT 623.04  ; RK_05 #2入壳吸盘破真空[A]
; rung 29
ILC(003)

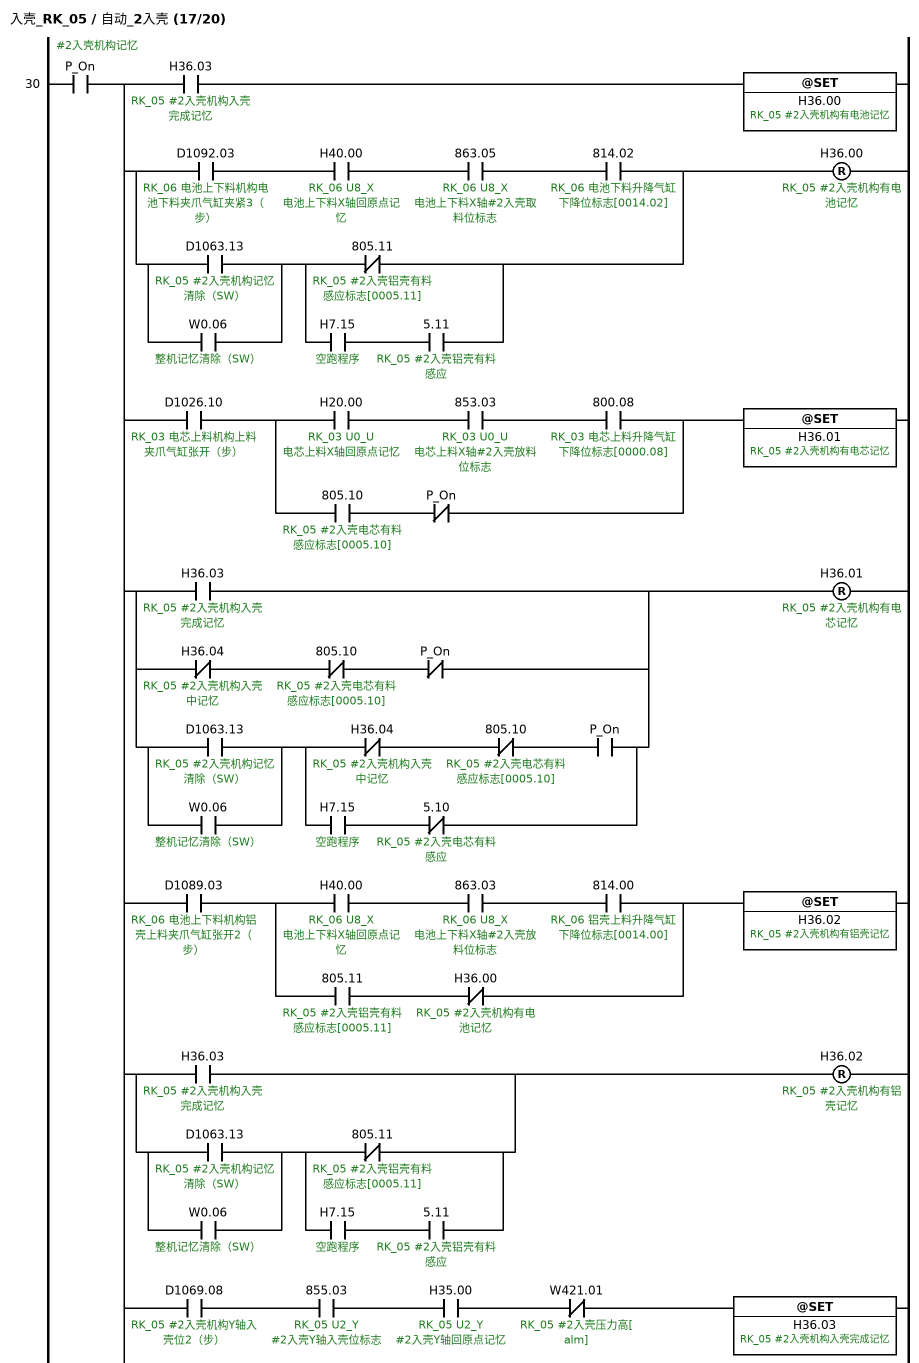

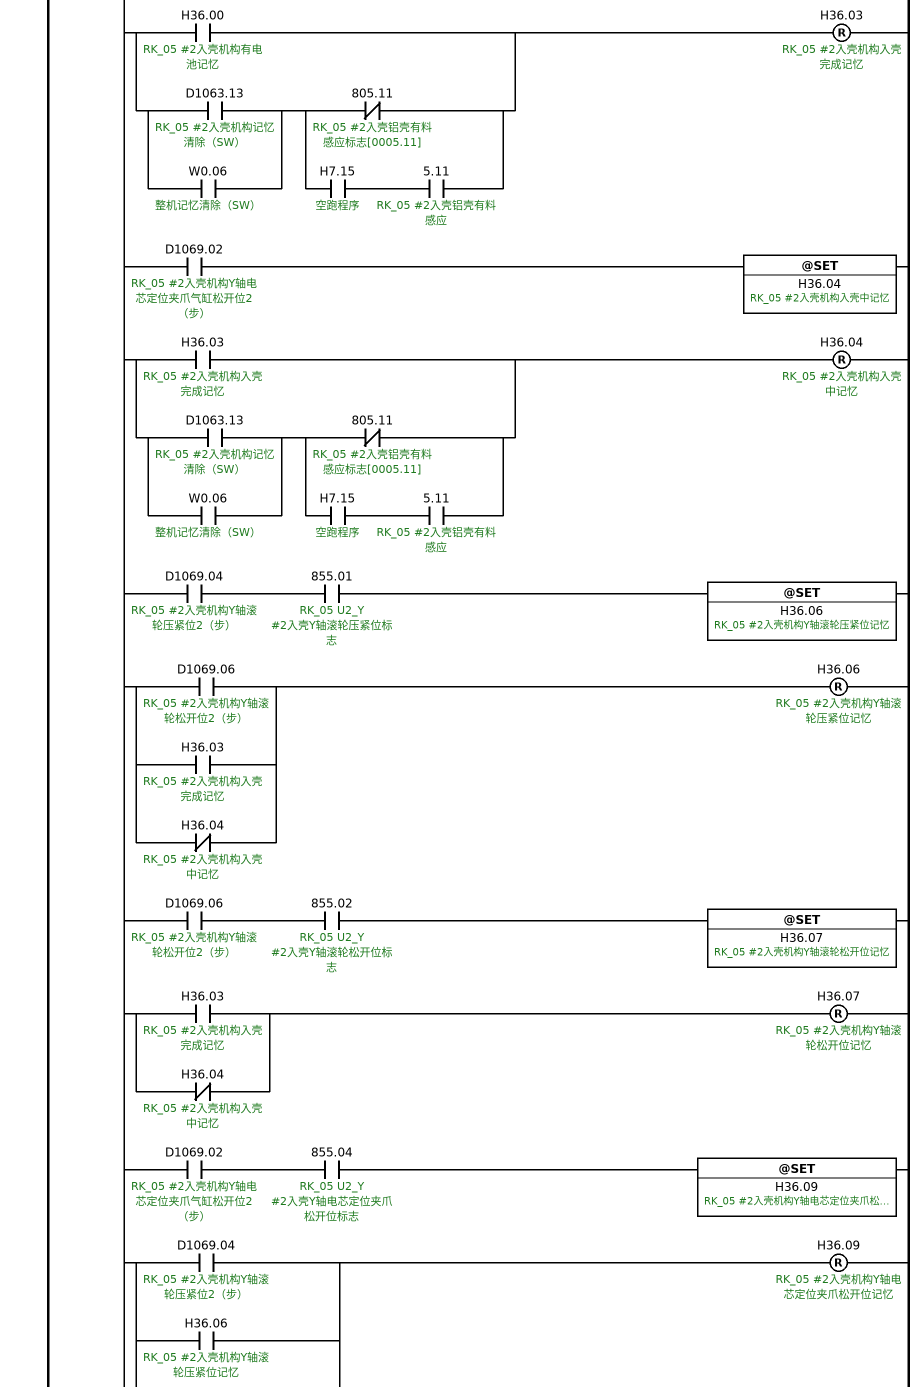

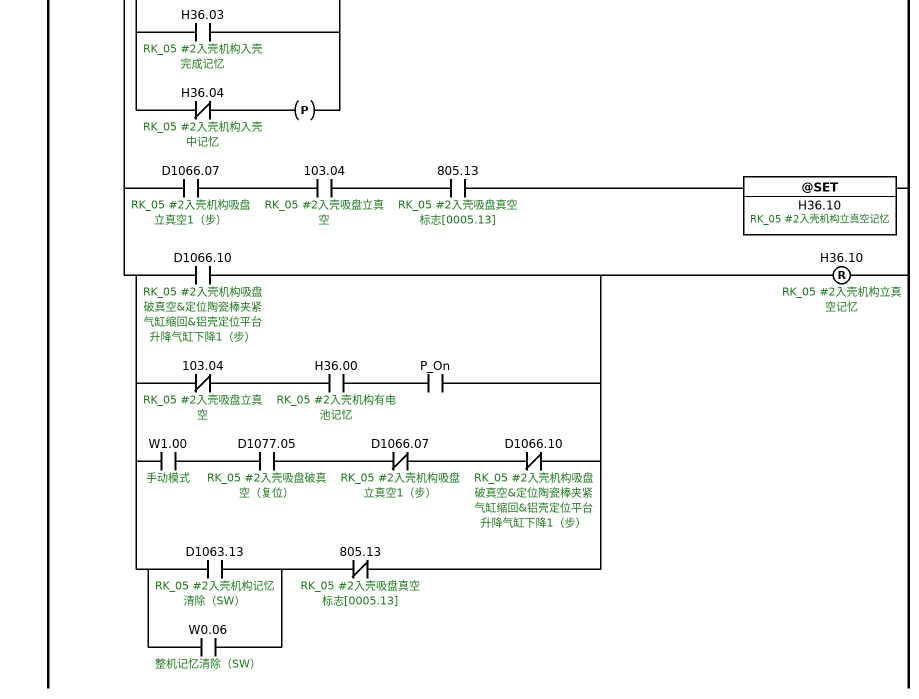
; rung 30: #2入壳机构记忆
LD P_On
OUT TR0
AND H36.03  ; RK_05 #2入壳机构入壳完成记忆
@SET H36.00  ; RK_05 #2入壳机构有电池记忆
LD TR0
LD D1092.03  ; RK_06 电池上下料机构电池下料夹爪气缸夹紧3（步）
AND H40.00  ; RK_06 U8_X 电池上下料X轴回原点记忆
AND 863.05  ; RK_06 U8_X 电池上下料X轴#2入壳取料位标志
AND 814.02  ; RK_06 电池下料升降气缸下降位标志[0014.02]
LD D1063.13  ; RK_05 #2入壳机构记忆清除（SW）
OR W0.06  ; 整机记忆清除（SW）
LDNOT 805.11  ; RK_05 #2入壳铝壳有料感应标志[0005.11]
LD H7.15  ; 空跑程序
AND 5.11  ; RK_05 #2入壳铝壳有料感应
ORLD
ANDLD
ORLD
ANDLD
RSET H36.00  ; RK_05 #2入壳机构有电池记忆
LD TR0
AND D1026.10  ; RK_03 电芯上料机构上料夹爪气缸张开（步）
LD H20.00  ; RK_03 U0_U 电芯上料X轴回原点记忆
AND 853.03  ; RK_03 U0_U 电芯上料X轴#2入壳放料位标志
AND 800.08  ; RK_03 电芯上料升降气缸下降位标志[0000.08]
LD 805.10  ; RK_05 #2入壳电芯有料感应标志[0005.10]
ANDNOT P_On
ORLD
ANDLD
@SET H36.01  ; RK_05 #2入壳机构有电芯记忆
LD TR0
LD H36.03  ; RK_05 #2入壳机构入壳完成记忆
LDNOT H36.04  ; RK_05 #2入壳机构入壳中记忆
ANDNOT 805.10  ; RK_05 #2入壳电芯有料感应标志[0005.10]
ANDNOT P_On
ORLD
LD D1063.13  ; RK_05 #2入壳机构记忆清除（SW）
OR W0.06  ; 整机记忆清除（SW）
LDNOT H36.04  ; RK_05 #2入壳机构入壳中记忆
ANDNOT 805.10  ; RK_05 #2入壳电芯有料感应标志[0005.10]
AND P_On
LD H7.15  ; 空跑程序
ANDNOT 5.10  ; RK_05 #2入壳电芯有料感应
ORLD
ANDLD
ORLD
ANDLD
RSET H36.01  ; RK_05 #2入壳机构有电芯记忆
LD TR0
AND D1089.03  ; RK_06 电池上下料机构铝壳上料夹爪气缸张开2（步）
LD H40.00  ; RK_06 U8_X 电池上下料X轴回原点记忆
AND 863.03  ; RK_06 U8_X 电池上下料X轴#2入壳放料位标志
AND 814.00  ; RK_06 铝壳上料升降气缸下降位标志[0014.00]
LD 805.11  ; RK_05 #2入壳铝壳有料感应标志[0005.11]
ANDNOT H36.00  ; RK_05 #2入壳机构有电池记忆
ORLD
ANDLD
@SET H36.02  ; RK_05 #2入壳机构有铝壳记忆
LD TR0
LD H36.03  ; RK_05 #2入壳机构入壳完成记忆
LD D1063.13  ; RK_05 #2入壳机构记忆清除（SW）
OR W0.06  ; 整机记忆清除（SW）
LDNOT 805.11  ; RK_05 #2入壳铝壳有料感应标志[0005.11]
LD H7.15  ; 空跑程序
AND 5.11  ; RK_05 #2入壳铝壳有料感应
ORLD
ANDLD
ORLD
ANDLD
RSET H36.02  ; RK_05 #2入壳机构有铝壳记忆
LD TR0
AND D1069.08  ; RK_05 #2入壳机构Y轴入壳位2（步）
AND 855.03  ; RK_05 U2_Y #2入壳Y轴入壳位标志
AND H35.00  ; RK_05 U2_Y #2入壳Y轴回原点记忆
ANDNOT W421.01  ; RK_05 #2入壳压力高[alm]
@SET H36.03  ; RK_05 #2入壳机构入壳完成记忆
LD TR0
LD H36.00  ; RK_05 #2入壳机构有电池记忆
LD D1063.13  ; RK_05 #2入壳机构记忆清除（SW）
OR W0.06  ; 整机记忆清除（SW）
LDNOT 805.11  ; RK_05 #2入壳铝壳有料感应标志[0005.11]
LD H7.15  ; 空跑程序
AND 5.11  ; RK_05 #2入壳铝壳有料感应
ORLD
ANDLD
ORLD
ANDLD
RSET H36.03  ; RK_05 #2入壳机构入壳完成记忆
LD TR0
AND D1069.02  ; RK_05 #2入壳机构Y轴电芯定位夹爪气缸松开位2（步）
@SET H36.04  ; RK_05 #2入壳机构入壳中记忆
LD TR0
LD H36.03  ; RK_05 #2入壳机构入壳完成记忆
LD D1063.13  ; RK_05 #2入壳机构记忆清除（SW）
OR W0.06  ; 整机记忆清除（SW）
LDNOT 805.11  ; RK_05 #2入壳铝壳有料感应标志[0005.11]
LD H7.15  ; 空跑程序
AND 5.11  ; RK_05 #2入壳铝壳有料感应
ORLD
ANDLD
ORLD
ANDLD
RSET H36.04  ; RK_05 #2入壳机构入壳中记忆
LD TR0
AND D1069.04  ; RK_05 #2入壳机构Y轴滚轮压紧位2（步）
AND 855.01  ; RK_05 U2_Y #2入壳Y轴滚轮压紧位标志
@SET H36.06  ; RK_05 #2入壳机构Y轴滚轮压紧位记忆
LD TR0
LD D1069.06  ; RK_05 #2入壳机构Y轴滚轮松开位2（步）
OR H36.03  ; RK_05 #2入壳机构入壳完成记忆
ORNOT H36.04  ; RK_05 #2入壳机构入壳中记忆
ANDLD
RSET H36.06  ; RK_05 #2入壳机构Y轴滚轮压紧位记忆
LD TR0
AND D1069.06  ; RK_05 #2入壳机构Y轴滚轮松开位2（步）
AND 855.02  ; RK_05 U2_Y #2入壳Y轴滚轮松开位标志
@SET H36.07  ; RK_05 #2入壳机构Y轴滚轮松开位记忆
LD TR0
LD H36.03  ; RK_05 #2入壳机构入壳完成记忆
ORNOT H36.04  ; RK_05 #2入壳机构入壳中记忆
ANDLD
RSET H36.07  ; RK_05 #2入壳机构Y轴滚轮松开位记忆
LD TR0
AND D1069.02  ; RK_05 #2入壳机构Y轴电芯定位夹爪气缸松开位2（步）
AND 855.04  ; RK_05 U2_Y #2入壳Y轴电芯定位夹爪松开位标志
@SET H36.09  ; RK_05 #2入壳机构Y轴电芯定位夹爪松开位记忆
LD TR0
LD D1069.04  ; RK_05 #2入壳机构Y轴滚轮压紧位2（步）
OR H36.06  ; RK_05 #2入壳机构Y轴滚轮压紧位记忆
OR H36.03  ; RK_05 #2入壳机构入壳完成记忆
LDNOT H36.04  ; RK_05 #2入壳机构入壳中记忆
UP(521)
ORLD
ANDLD
RSET H36.09  ; RK_05 #2入壳机构Y轴电芯定位夹爪松开位记忆
LD TR0
AND D1066.07  ; RK_05 #2入壳机构吸盘立真空1（步）
AND 103.04  ; RK_05 #2入壳吸盘立真空
AND 805.13  ; RK_05 #2入壳吸盘真空标志[0005.13]
@SET H36.10  ; RK_05 #2入壳机构立真空记忆
LD TR0
LD D1066.10  ; RK_05 #2入壳机构吸盘破真空&定位陶瓷棒夹紧气缸缩回&铝壳定位平台升降气缸下降1（步）
LDNOT 103.04  ; RK_05 #2入壳吸盘立真空
AND H36.00  ; RK_05 #2入壳机构有电池记忆
AND P_On
ORLD
LD W1.00  ; 手动模式  // 20181116新增
AND D1077.05  ; RK_05 #2入壳吸盘破真空（复位）
ANDNOT D1066.07  ; RK_05 #2入壳机构吸盘立真空1（步）
ANDNOT D1066.10  ; RK_05 #2入壳机构吸盘破真空&定位陶瓷棒夹紧气缸缩回&铝壳定位平台升降气缸下降1（步）
ORLD
LD D1063.13  ; RK_05 #2入壳机构记忆清除（SW）
OR W0.06  ; 整机记忆清除（SW）
ANDNOT 805.13  ; RK_05 #2入壳吸盘真空标志[0005.13]
ORLD
ANDLD
RSET H36.10  ; RK_05 #2入壳机构立真空记忆

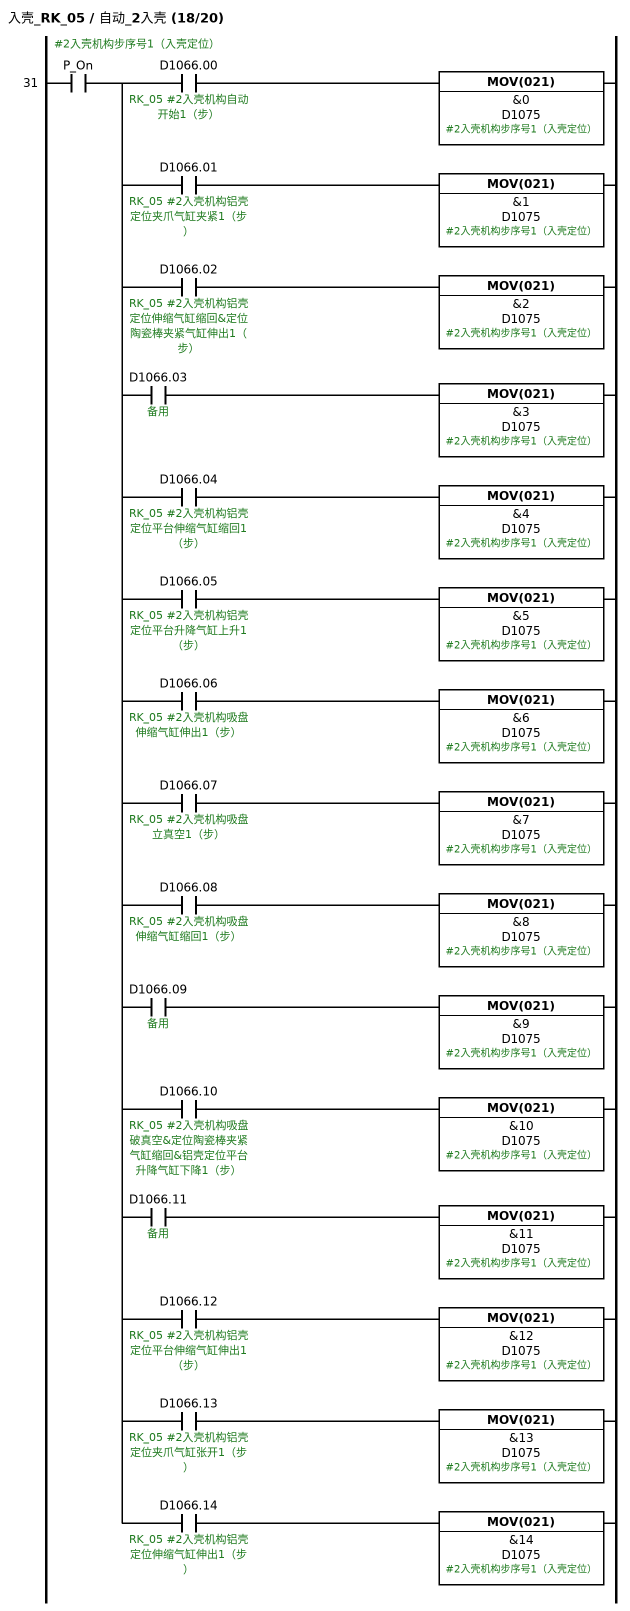
; rung 31: #2入壳机构步序号1（入壳定位）
LD P_On
OUT TR0
AND D1066.00  ; RK_05 #2入壳机构自动开始1（步）
MOV(021) &0 D1075  ; #2入壳机构步序号1（入壳定位）
LD TR0
AND D1066.01  ; RK_05 #2入壳机构铝壳定位夹爪气缸夹紧1（步）
MOV(021) &1 D1075  ; #2入壳机构步序号1（入壳定位）
LD TR0
AND D1066.02  ; RK_05 #2入壳机构铝壳定位伸缩气缸缩回&定位陶瓷棒夹紧气缸伸出1（步）
MOV(021) &2 D1075  ; #2入壳机构步序号1（入壳定位）
LD TR0
AND D1066.03  ; 备用
MOV(021) &3 D1075  ; #2入壳机构步序号1（入壳定位）
LD TR0
AND D1066.04  ; RK_05 #2入壳机构铝壳定位平台伸缩气缸缩回1（步）
MOV(021) &4 D1075  ; #2入壳机构步序号1（入壳定位）
LD TR0
AND D1066.05  ; RK_05 #2入壳机构铝壳定位平台升降气缸上升1（步）
MOV(021) &5 D1075  ; #2入壳机构步序号1（入壳定位）
LD TR0
AND D1066.06  ; RK_05 #2入壳机构吸盘伸缩气缸伸出1（步）
MOV(021) &6 D1075  ; #2入壳机构步序号1（入壳定位）
LD TR0
AND D1066.07  ; RK_05 #2入壳机构吸盘立真空1（步）
MOV(021) &7 D1075  ; #2入壳机构步序号1（入壳定位）
LD TR0
AND D1066.08  ; RK_05 #2入壳机构吸盘伸缩气缸缩回1（步）
MOV(021) &8 D1075  ; #2入壳机构步序号1（入壳定位）
LD TR0
AND D1066.09  ; 备用
MOV(021) &9 D1075  ; #2入壳机构步序号1（入壳定位）
LD TR0
AND D1066.10  ; RK_05 #2入壳机构吸盘破真空&定位陶瓷棒夹紧气缸缩回&铝壳定位平台升降气缸下降1（步）
MOV(021) &10 D1075  ; #2入壳机构步序号1（入壳定位）
LD TR0
AND D1066.11  ; 备用
MOV(021) &11 D1075  ; #2入壳机构步序号1（入壳定位）
LD TR0
AND D1066.12  ; RK_05 #2入壳机构铝壳定位平台伸缩气缸伸出1（步）
MOV(021) &12 D1075  ; #2入壳机构步序号1（入壳定位）
LD TR0
AND D1066.13  ; RK_05 #2入壳机构铝壳定位夹爪气缸张开1（步）
MOV(021) &13 D1075  ; #2入壳机构步序号1（入壳定位）
LD TR0
AND D1066.14  ; RK_05 #2入壳机构铝壳定位伸缩气缸伸出1（步）
MOV(021) &14 D1075  ; #2入壳机构步序号1（入壳定位）

